    |   movel([0.078731, -1.406852, -2.551684, -0.753853, 1.570796, 1.649527],accel_mss,speed_ms,0,blend_radius_m)
    |   movel([0.077871, -1.407087, -2.551509, -0.753793, 1.570796, 1.648667],accel_mss,speed_ms,0,blend_radius_m)
    |   movel([0.077016, -1.407341, -2.551319, -0.753728, 1.570796, 1.647812],accel_mss,speed_ms,0,blend_radius_m)
    |   movel([0.076261, -1.407587, -2.551136, -0.753666, 1.570796, 1.647058],accel_mss,speed_ms,0,blend_radius_m)
    |   movel([0.075139, -1.407960, -2.550859, -0.753571, 1.570796, 1.645936],accel_mss,speed_ms,0,blend_radius_m)
    |   speed_ms = 0.003
    |   movel([0.075139, -1.411176, -2.552300, -0.748913, 1.570796, 1.645936],accel_mss,speed_ms,0,blend_radius_m)
    |   speed_ms = 0.007
    |   movel([0.074668, -1.411273, -2.552227, -0.748889, 1.570796, 1.645464],accel_mss,speed_ms,0,blend_radius_m)
    |   movel([0.074481, -1.411194, -2.552286, -0.748909, 1.570796, 1.645278],accel_mss,speed_ms,0,blend_radius_m)
    |   movel([0.074467, -1.410958, -2.552463, -0.748968, 1.570796, 1.645263],accel_mss,speed_ms,0,blend_radius_m)
    |   movel([0.074692, -1.410622, -2.552715, -0.749052, 1.570796, 1.645489],accel_mss,speed_ms,0,blend_radius_m)
    |   movel([0.075140, -1.410315, -2.552945, -0.749129, 1.570796, 1.645937],accel_mss,speed_ms,0,blend_radius_m)
    |   movel([0.075912, -1.409983, -2.553193, -0.749213, 1.570796, 1.646708],accel_mss,speed_ms,0,blend_radius_m)
    |   movel([0.077256, -1.409535, -2.553528, -0.749326, 1.570796, 1.648052],accel_mss,speed_ms,0,blend_radius_m)
    |   movel([0.078806, -1.409077, -2.553870, -0.749442, 1.570796, 1.649603],accel_mss,speed_ms,0,blend_radius_m)
    |   movel([0.079979, -1.408805, -2.554073, -0.749511, 1.570796, 1.650775],accel_mss,speed_ms,0,blend_radius_m)
    |   movel([0.080824, -1.408690, -2.554159, -0.749540, 1.570796, 1.651621],accel_mss,speed_ms,0,blend_radius_m)
    |   movel([0.081268, -1.408772, -2.554098, -0.749519, 1.570796, 1.652064],accel_mss,speed_ms,0,blend_radius_m)
    |   movel([0.081447, -1.408903, -2.554000, -0.749486, 1.570796, 1.652243],accel_mss,speed_ms,0,blend_radius_m)
    |   movel([0.081473, -1.409173, -2.553798, -0.749418, 1.570796, 1.652269],accel_mss,speed_ms,0,blend_radius_m)
    |   movel([0.081179, -1.409435, -2.553602, -0.749351, 1.570796, 1.651975],accel_mss,speed_ms,0,blend_radius_m)
    |   movel([0.080823, -1.409552, -2.553515, -0.749322, 1.570796, 1.651619],accel_mss,speed_ms,0,blend_radius_m)
    |   movel([0.080297, -1.409695, -2.553409, -0.749286, 1.570796, 1.651093],accel_mss,speed_ms,0,blend_radius_m)
    |   movel([0.079504, -1.409881, -2.553270, -0.749239, 1.570796, 1.650301],accel_mss,speed_ms,0,blend_radius_m)
    |   movel([0.078731, -1.410072, -2.553127, -0.749191, 1.570796, 1.649527],accel_mss,speed_ms,0,blend_radius_m)
    |   movel([0.077871, -1.410306, -2.552951, -0.749132, 1.570796, 1.648667],accel_mss,speed_ms,0,blend_radius_m)
    |   movel([0.077016, -1.410560, -2.552762, -0.749068, 1.570796, 1.647812],accel_mss,speed_ms,0,blend_radius_m)
    |   movel([0.076261, -1.410805, -2.552578, -0.749006, 1.570796, 1.647058],accel_mss,speed_ms,0,blend_radius_m)
    |   movel([0.075139, -1.411176, -2.552300, -0.748913, 1.570796, 1.645936],accel_mss,speed_ms,0,blend_radius_m)
    |   speed_ms = 0.003
    |   movel([0.075139, -1.398436, -2.546485, -0.767469, 1.570796, 1.645936],accel_mss,speed_ms,0,blend_radius_m)
    |   speed_ms = 1.000
    |   movel([0.075139, -1.373952, -2.534460, -0.803977, 1.570796, 1.645936],accel_mss,speed_ms,0,blend_radius_m)
    |   movel([0.075519, -1.372021, -2.535826, -0.804542, 1.570796, 1.646315],accel_mss,speed_ms,0,blend_radius_m)
    |   movel([0.075519, -1.396541, -2.547875, -0.767973, 1.570796, 1.646315],accel_mss,speed_ms,0,blend_radius_m)
    |   speed_ms = 0.003
    |   movel([0.075519, -1.406080, -2.552258, -0.754051, 1.570796, 1.646315],accel_mss,speed_ms,0,blend_radius_m)
    |   speed_ms = 0.007
    |   movel([0.075126, -1.406076, -2.552261, -0.754052, 1.570796, 1.645923],accel_mss,speed_ms,0,blend_radius_m)
    |   movel([0.074945, -1.405955, -2.552351, -0.754083, 1.570796, 1.645741],accel_mss,speed_ms,0,blend_radius_m)
    |   movel([0.074905, -1.405527, -2.552669, -0.754193, 1.570796, 1.645701],accel_mss,speed_ms,0,blend_radius_m)
    |   movel([0.074901, -1.405141, -2.552955, -0.754293, 1.570796, 1.645697],accel_mss,speed_ms,0,blend_radius_m)
    |   movel([0.074910, -1.404710, -2.553275, -0.754404, 1.570796, 1.645707],accel_mss,speed_ms,0,blend_radius_m)
    |   movel([0.074938, -1.404075, -2.553745, -0.754569, 1.570796, 1.645734],accel_mss,speed_ms,0,blend_radius_m)
    |   movel([0.074975, -1.403788, -2.553958, -0.754644, 1.570796, 1.645771],accel_mss,speed_ms,0,blend_radius_m)
    |   movel([0.075148, -1.403554, -2.554131, -0.754705, 1.570796, 1.645944],accel_mss,speed_ms,0,blend_radius_m)
    |   movel([0.075346, -1.403676, -2.554040, -0.754673, 1.570796, 1.646142],accel_mss,speed_ms,0,blend_radius_m)
    |   movel([0.075432, -1.403876, -2.553893, -0.754621, 1.570796, 1.646229],accel_mss,speed_ms,0,blend_radius_m)
    |   movel([0.075542, -1.404111, -2.553718, -0.754559, 1.570796, 1.646338],accel_mss,speed_ms,0,blend_radius_m)
    |   movel([0.075676, -1.404370, -2.553527, -0.754492, 1.570796, 1.646472],accel_mss,speed_ms,0,blend_radius_m)
    |   movel([0.075914, -1.404778, -2.553224, -0.754387, 1.570796, 1.646711],accel_mss,speed_ms,0,blend_radius_m)
    |   movel([0.076091, -1.404951, -2.553096, -0.754342, 1.570796, 1.646887],accel_mss,speed_ms,0,blend_radius_m)
    |   movel([0.076338, -1.405044, -2.553027, -0.754318, 1.570796, 1.647135],accel_mss,speed_ms,0,blend_radius_m)
    |   movel([0.076878, -1.405129, -2.552964, -0.754296, 1.570796, 1.647674],accel_mss,speed_ms,0,blend_radius_m)
    |   movel([0.077216, -1.405165, -2.552937, -0.754286, 1.570796, 1.648012],accel_mss,speed_ms,0,blend_radius_m)
    |   movel([0.077528, -1.405191, -2.552918, -0.754280, 1.570796, 1.648324],accel_mss,speed_ms,0,blend_radius_m)
    |   movel([0.077792, -1.405202, -2.552910, -0.754277, 1.570796, 1.648589],accel_mss,speed_ms,0,blend_radius_m)
    |   movel([0.078078, -1.405163, -2.552939, -0.754287, 1.570796, 1.648874],accel_mss,speed_ms,0,blend_radius_m)
    |   movel([0.078293, -1.405186, -2.552922, -0.754281, 1.570796, 1.649090],accel_mss,speed_ms,0,blend_radius_m)
    |   movel([0.078458, -1.405300, -2.552837, -0.754252, 1.570796, 1.649254],accel_mss,speed_ms,0,blend_radius_m)
    |   movel([0.078022, -1.405459, -2.552719, -0.754211, 1.570796, 1.648818],accel_mss,speed_ms,0,blend_radius_m)
    |   movel([0.077584, -1.405591, -2.552621, -0.754177, 1.570796, 1.648380],accel_mss,speed_ms,0,blend_radius_m)
    |   movel([0.077076, -1.405736, -2.552513, -0.754139, 1.570796, 1.647873],accel_mss,speed_ms,0,blend_radius_m)
    |   movel([0.076136, -1.405975, -2.552336, -0.754078, 1.570796, 1.646933],accel_mss,speed_ms,0,blend_radius_m)
    |   movel([0.075519, -1.406080, -2.552258, -0.754051, 1.570796, 1.646315],accel_mss,speed_ms,0,blend_radius_m)
    |   speed_ms = 0.003
    |   movel([0.075519, -1.409302, -2.553702, -0.749385, 1.570796, 1.646315],accel_mss,speed_ms,0,blend_radius_m)
    |   speed_ms = 0.007
    |   movel([0.075126, -1.409298, -2.553705, -0.749386, 1.570796, 1.645923],accel_mss,speed_ms,0,blend_radius_m)
    |   movel([0.074945, -1.409177, -2.553795, -0.749417, 1.570796, 1.645741],accel_mss,speed_ms,0,blend_radius_m)
    |   movel([0.074905, -1.408750, -2.554114, -0.749525, 1.570796, 1.645701],accel_mss,speed_ms,0,blend_radius_m)
    |   movel([0.074901, -1.408365, -2.554401, -0.749623, 1.570796, 1.645697],accel_mss,speed_ms,0,blend_radius_m)
    |   movel([0.074910, -1.407935, -2.554721, -0.749732, 1.570796, 1.645707],accel_mss,speed_ms,0,blend_radius_m)
    |   movel([0.074938, -1.407303, -2.555192, -0.749894, 1.570796, 1.645734],accel_mss,speed_ms,0,blend_radius_m)
    |   movel([0.074975, -1.407016, -2.555406, -0.749967, 1.570796, 1.645771],accel_mss,speed_ms,0,blend_radius_m)
    |   movel([0.075148, -1.406782, -2.555579, -0.750027, 1.570796, 1.645944],accel_mss,speed_ms,0,blend_radius_m)
    |   movel([0.075346, -1.406905, -2.555488, -0.749996, 1.570796, 1.646142],accel_mss,speed_ms,0,blend_radius_m)
    |   movel([0.075432, -1.407104, -2.555340, -0.749945, 1.570796, 1.646229],accel_mss,speed_ms,0,blend_radius_m)
    |   movel([0.075542, -1.407338, -2.555166, -0.749885, 1.570796, 1.646338],accel_mss,speed_ms,0,blend_radius_m)
    |   movel([0.075676, -1.407596, -2.554974, -0.749819, 1.570796, 1.646472],accel_mss,speed_ms,0,blend_radius_m)
    |   movel([0.075914, -1.408003, -2.554671, -0.749715, 1.570796, 1.646711],accel_mss,speed_ms,0,blend_radius_m)
    |   movel([0.076091, -1.408176, -2.554542, -0.749671, 1.570796, 1.646887],accel_mss,speed_ms,0,blend_radius_m)
    |   movel([0.076338, -1.408268, -2.554473, -0.749647, 1.570796, 1.647135],accel_mss,speed_ms,0,blend_radius_m)
    |   movel([0.076878, -1.408353, -2.554410, -0.749626, 1.570796, 1.647674],accel_mss,speed_ms,0,blend_radius_m)
    |   movel([0.077216, -1.408390, -2.554383, -0.749616, 1.570796, 1.648012],accel_mss,speed_ms,0,blend_radius_m)
    |   movel([0.077528, -1.408415, -2.554364, -0.749610, 1.570796, 1.648324],accel_mss,speed_ms,0,blend_radius_m)
    |   movel([0.077792, -1.408426, -2.554356, -0.749607, 1.570796, 1.648589],accel_mss,speed_ms,0,blend_radius_m)
    |   movel([0.078078, -1.408387, -2.554385, -0.749617, 1.570796, 1.648874],accel_mss,speed_ms,0,blend_radius_m)
    |   movel([0.078293, -1.408410, -2.554368, -0.749611, 1.570796, 1.649090],accel_mss,speed_ms,0,blend_radius_m)
    |   movel([0.078458, -1.408524, -2.554282, -0.749582, 1.570796, 1.649254],accel_mss,speed_ms,0,blend_radius_m)
    |   movel([0.078022, -1.408683, -2.554164, -0.749542, 1.570796, 1.648818],accel_mss,speed_ms,0,blend_radius_m)
    |   movel([0.077584, -1.408814, -2.554067, -0.749509, 1.570796, 1.648380],accel_mss,speed_ms,0,blend_radius_m)
    |   movel([0.077076, -1.408959, -2.553958, -0.749472, 1.570796, 1.647873],accel_mss,speed_ms,0,blend_radius_m)
    |   movel([0.076136, -1.409198, -2.553780, -0.749411, 1.570796, 1.646933],accel_mss,speed_ms,0,blend_radius_m)
    |   movel([0.075519, -1.409302, -2.553702, -0.749385, 1.570796, 1.646315],accel_mss,speed_ms,0,blend_radius_m)
    |   speed_ms = 0.003
    |   movel([0.075519, -1.396541, -2.547875, -0.767973, 1.570796, 1.646315],accel_mss,speed_ms,0,blend_radius_m)
    |   speed_ms = 1.000
    |   movel([0.075519, -1.372021, -2.535826, -0.804542, 1.570796, 1.646315],accel_mss,speed_ms,0,blend_radius_m)
    |   movel([0.077083, -1.370467, -2.536922, -0.805000, 1.570796, 1.647879],accel_mss,speed_ms,0,blend_radius_m)
    |   movel([0.077083, -1.395016, -2.548990, -0.768383, 1.570796, 1.647879],accel_mss,speed_ms,0,blend_radius_m)
    |   speed_ms = 0.003
    |   movel([0.077083, -1.404567, -2.553381, -0.754441, 1.570796, 1.647879],accel_mss,speed_ms,0,blend_radius_m)
    |   speed_ms = 0.007
    |   movel([0.076403, -1.404193, -2.553658, -0.754538, 1.570796, 1.647199],accel_mss,speed_ms,0,blend_radius_m)
    |   movel([0.076021, -1.403445, -2.554211, -0.754733, 1.570796, 1.646818],accel_mss,speed_ms,0,blend_radius_m)
    |   movel([0.075316, -1.401677, -2.555516, -0.755196, 1.570796, 1.646112],accel_mss,speed_ms,0,blend_radius_m)
    |   movel([0.074634, -1.399869, -2.556846, -0.755675, 1.570796, 1.645431],accel_mss,speed_ms,0,blend_radius_m)
    |   movel([0.074243, -1.398639, -2.557747, -0.756003, 1.570796, 1.645039],accel_mss,speed_ms,0,blend_radius_m)
    |   movel([0.074191, -1.398445, -2.557889, -0.756055, 1.570796, 1.644987],accel_mss,speed_ms,0,blend_radius_m)
    |   movel([0.074083, -1.398061, -2.558171, -0.756158, 1.570796, 1.644879],accel_mss,speed_ms,0,blend_radius_m)
    |   movel([0.073955, -1.397607, -2.558503, -0.756280, 1.570796, 1.644752],accel_mss,speed_ms,0,blend_radius_m)
    |   movel([0.073822, -1.397131, -2.558850, -0.756408, 1.570796, 1.644618],accel_mss,speed_ms,0,blend_radius_m)
    |   movel([0.073030, -1.393944, -2.561169, -0.757276, 1.570796, 1.643826],accel_mss,speed_ms,0,blend_radius_m)
    |   movel([0.072490, -1.390932, -2.563348, -0.758110, 1.570796, 1.643286],accel_mss,speed_ms,0,blend_radius_m)
    |   movel([0.072193, -1.387994, -2.565460, -0.758936, 1.570796, 1.642990],accel_mss,speed_ms,0,blend_radius_m)
    |   movel([0.072126, -1.385031, -2.567577, -0.759781, 1.570796, 1.642923],accel_mss,speed_ms,0,blend_radius_m)
    |   movel([0.072151, -1.383881, -2.568396, -0.760113, 1.570796, 1.642947],accel_mss,speed_ms,0,blend_radius_m)
    |   movel([0.072187, -1.383304, -2.568805, -0.760280, 1.570796, 1.642984],accel_mss,speed_ms,0,blend_radius_m)
    |   movel([0.072246, -1.382955, -2.569053, -0.760381, 1.570796, 1.643042],accel_mss,speed_ms,0,blend_radius_m)
    |   movel([0.072513, -1.382648, -2.569271, -0.760471, 1.570796, 1.643309],accel_mss,speed_ms,0,blend_radius_m)
    |   movel([0.073127, -1.382500, -2.569376, -0.760513, 1.570796, 1.643923],accel_mss,speed_ms,0,blend_radius_m)
    |   movel([0.073892, -1.382409, -2.569440, -0.760540, 1.570796, 1.644689],accel_mss,speed_ms,0,blend_radius_m)
    |   movel([0.079022, -1.381656, -2.569973, -0.760760, 1.570796, 1.649818],accel_mss,speed_ms,0,blend_radius_m)
    |   movel([0.084810, -1.380457, -2.570821, -0.761111, 1.570796, 1.655606],accel_mss,speed_ms,0,blend_radius_m)
    |   movel([0.090456, -1.379003, -2.571845, -0.761540, 1.570796, 1.661253],accel_mss,speed_ms,0,blend_radius_m)
    |   movel([0.095111, -1.377468, -2.572924, -0.761997, 1.570796, 1.665908],accel_mss,speed_ms,0,blend_radius_m)
    |   movel([0.097708, -1.376448, -2.573639, -0.762302, 1.570796, 1.668504],accel_mss,speed_ms,0,blend_radius_m)
    |   movel([0.100378, -1.375309, -2.574435, -0.762644, 1.570796, 1.671174],accel_mss,speed_ms,0,blend_radius_m)
    |   movel([0.102904, -1.374151, -2.575243, -0.762994, 1.570796, 1.673700],accel_mss,speed_ms,0,blend_radius_m)
    |   movel([0.105045, -1.373074, -2.575993, -0.763322, 1.570796, 1.675841],accel_mss,speed_ms,0,blend_radius_m)
    |   movel([0.105543, -1.372819, -2.576171, -0.763400, 1.570796, 1.676340],accel_mss,speed_ms,0,blend_radius_m)
    |   movel([0.105878, -1.372668, -2.576275, -0.763446, 1.570796, 1.676675],accel_mss,speed_ms,0,blend_radius_m)
    |   movel([0.106228, -1.372598, -2.576324, -0.763467, 1.570796, 1.677024],accel_mss,speed_ms,0,blend_radius_m)
    |   movel([0.106336, -1.372808, -2.576178, -0.763403, 1.570796, 1.677133],accel_mss,speed_ms,0,blend_radius_m)
    |   movel([0.106198, -1.374131, -2.575258, -0.763001, 1.570796, 1.676995],accel_mss,speed_ms,0,blend_radius_m)
    |   movel([0.105975, -1.375739, -2.574135, -0.762515, 1.570796, 1.676771],accel_mss,speed_ms,0,blend_radius_m)
    |   movel([0.105644, -1.377653, -2.572794, -0.761942, 1.570796, 1.676440],accel_mss,speed_ms,0,blend_radius_m)
    |   movel([0.104699, -1.381947, -2.569767, -0.760675, 1.570796, 1.675495],accel_mss,speed_ms,0,blend_radius_m)
    |   movel([0.103481, -1.386121, -2.566799, -0.759469, 1.570796, 1.674277],accel_mss,speed_ms,0,blend_radius_m)
    |   movel([0.102014, -1.390127, -2.563928, -0.758335, 1.570796, 1.672810],accel_mss,speed_ms,0,blend_radius_m)
    |   movel([0.100315, -1.393925, -2.561183, -0.757281, 1.570796, 1.671111],accel_mss,speed_ms,0,blend_radius_m)
    |   movel([0.099682, -1.395155, -2.560289, -0.756944, 1.570796, 1.670478],accel_mss,speed_ms,0,blend_radius_m)
    |   movel([0.098968, -1.396436, -2.559357, -0.756596, 1.570796, 1.669764],accel_mss,speed_ms,0,blend_radius_m)
    |   movel([0.098297, -1.397567, -2.558532, -0.756291, 1.570796, 1.669093],accel_mss,speed_ms,0,blend_radius_m)
    |   movel([0.097942, -1.398033, -2.558191, -0.756165, 1.570796, 1.668739],accel_mss,speed_ms,0,blend_radius_m)
    |   movel([0.097526, -1.398382, -2.557935, -0.756072, 1.570796, 1.668322],accel_mss,speed_ms,0,blend_radius_m)
    |   movel([0.096641, -1.398930, -2.557534, -0.755925, 1.570796, 1.667437],accel_mss,speed_ms,0,blend_radius_m)
    |   movel([0.095567, -1.399532, -2.557093, -0.755764, 1.570796, 1.666363],accel_mss,speed_ms,0,blend_radius_m)
    |   movel([0.094415, -1.400113, -2.556666, -0.755610, 1.570796, 1.665211],accel_mss,speed_ms,0,blend_radius_m)
    |   movel([0.091915, -1.401217, -2.555855, -0.755317, 1.570796, 1.662711],accel_mss,speed_ms,0,blend_radius_m)
    |   movel([0.089053, -1.402291, -2.555063, -0.755035, 1.570796, 1.659849],accel_mss,speed_ms,0,blend_radius_m)
    |   movel([0.086165, -1.403221, -2.554377, -0.754791, 1.570796, 1.656961],accel_mss,speed_ms,0,blend_radius_m)
    |   movel([0.083581, -1.403891, -2.553881, -0.754617, 1.570796, 1.654377],accel_mss,speed_ms,0,blend_radius_m)
    |   movel([0.080960, -1.404386, -2.553515, -0.754488, 1.570796, 1.651756],accel_mss,speed_ms,0,blend_radius_m)
    |   movel([0.078742, -1.404605, -2.553352, -0.754431, 1.570796, 1.649539],accel_mss,speed_ms,0,blend_radius_m)
    |   movel([0.077083, -1.404567, -2.553381, -0.754441, 1.570796, 1.647879],accel_mss,speed_ms,0,blend_radius_m)
    |   speed_ms = 0.003
    |   movel([0.077083, -1.407793, -2.554827, -0.749769, 1.570796, 1.647879],accel_mss,speed_ms,0,blend_radius_m)
    |   speed_ms = 0.007
    |   movel([0.076403, -1.407420, -2.555105, -0.749864, 1.570796, 1.647199],accel_mss,speed_ms,0,blend_radius_m)
    |   movel([0.076021, -1.406674, -2.555660, -0.750055, 1.570796, 1.646818],accel_mss,speed_ms,0,blend_radius_m)
    |   movel([0.075316, -1.404911, -2.556967, -0.750510, 1.570796, 1.646112],accel_mss,speed_ms,0,blend_radius_m)
    |   movel([0.074634, -1.403108, -2.558300, -0.750981, 1.570796, 1.645431],accel_mss,speed_ms,0,blend_radius_m)
    |   movel([0.074243, -1.401882, -2.559203, -0.751304, 1.570796, 1.645039],accel_mss,speed_ms,0,blend_radius_m)
    |   movel([0.074191, -1.401688, -2.559346, -0.751355, 1.570796, 1.644987],accel_mss,speed_ms,0,blend_radius_m)
    |   movel([0.074083, -1.401305, -2.559628, -0.751456, 1.570796, 1.644879],accel_mss,speed_ms,0,blend_radius_m)
    |   movel([0.073955, -1.400852, -2.559960, -0.751576, 1.570796, 1.644752],accel_mss,speed_ms,0,blend_radius_m)
    |   movel([0.073822, -1.400378, -2.560308, -0.751702, 1.570796, 1.644618],accel_mss,speed_ms,0,blend_radius_m)
    |   movel([0.073030, -1.397200, -2.562633, -0.752556, 1.570796, 1.643826],accel_mss,speed_ms,0,blend_radius_m)
    |   movel([0.072490, -1.394196, -2.564816, -0.753377, 1.570796, 1.643286],accel_mss,speed_ms,0,blend_radius_m)
    |   movel([0.072193, -1.391266, -2.566933, -0.754190, 1.570796, 1.642990],accel_mss,speed_ms,0,blend_radius_m)
    |   movel([0.072126, -1.388311, -2.569056, -0.755023, 1.570796, 1.642923],accel_mss,speed_ms,0,blend_radius_m)
    |   movel([0.072151, -1.387164, -2.569876, -0.755349, 1.570796, 1.642947],accel_mss,speed_ms,0,blend_radius_m)
    |   movel([0.072187, -1.386589, -2.570287, -0.755514, 1.570796, 1.642984],accel_mss,speed_ms,0,blend_radius_m)
    |   movel([0.072246, -1.386241, -2.570535, -0.755613, 1.570796, 1.643042],accel_mss,speed_ms,0,blend_radius_m)
    |   movel([0.072513, -1.385934, -2.570753, -0.755701, 1.570796, 1.643309],accel_mss,speed_ms,0,blend_radius_m)
    |   movel([0.073127, -1.385787, -2.570858, -0.755744, 1.570796, 1.643923],accel_mss,speed_ms,0,blend_radius_m)
    |   movel([0.073892, -1.385697, -2.570922, -0.755770, 1.570796, 1.644689],accel_mss,speed_ms,0,blend_radius_m)
    |   movel([0.079022, -1.384945, -2.571457, -0.755986, 1.570796, 1.649818],accel_mss,speed_ms,0,blend_radius_m)
    |   movel([0.084810, -1.383749, -2.572307, -0.756333, 1.570796, 1.655606],accel_mss,speed_ms,0,blend_radius_m)
    |   movel([0.090456, -1.382300, -2.573334, -0.756755, 1.570796, 1.661253],accel_mss,speed_ms,0,blend_radius_m)
    |   movel([0.095111, -1.380769, -2.574415, -0.757205, 1.570796, 1.665908],accel_mss,speed_ms,0,blend_radius_m)
    |   movel([0.097708, -1.379752, -2.575132, -0.757506, 1.570796, 1.668504],accel_mss,speed_ms,0,blend_radius_m)
    |   movel([0.100378, -1.378616, -2.575930, -0.757843, 1.570796, 1.671174],accel_mss,speed_ms,0,blend_radius_m)
    |   movel([0.102904, -1.377461, -2.576739, -0.758188, 1.570796, 1.673700],accel_mss,speed_ms,0,blend_radius_m)
    |   movel([0.105045, -1.376387, -2.577491, -0.758511, 1.570796, 1.675841],accel_mss,speed_ms,0,blend_radius_m)
    |   movel([0.105543, -1.376132, -2.577669, -0.758588, 1.570796, 1.676340],accel_mss,speed_ms,0,blend_radius_m)
    |   movel([0.105878, -1.375982, -2.577774, -0.758633, 1.570796, 1.676675],accel_mss,speed_ms,0,blend_radius_m)
    |   movel([0.106228, -1.375912, -2.577822, -0.758654, 1.570796, 1.677024],accel_mss,speed_ms,0,blend_radius_m)
    |   movel([0.106336, -1.376121, -2.577677, -0.758591, 1.570796, 1.677133],accel_mss,speed_ms,0,blend_radius_m)
    |   movel([0.106198, -1.377441, -2.576754, -0.758194, 1.570796, 1.676995],accel_mss,speed_ms,0,blend_radius_m)
    |   movel([0.105975, -1.379044, -2.575629, -0.757716, 1.570796, 1.676771],accel_mss,speed_ms,0,blend_radius_m)
    |   movel([0.105644, -1.380953, -2.574285, -0.757151, 1.570796, 1.676440],accel_mss,speed_ms,0,blend_radius_m)
    |   movel([0.104699, -1.385235, -2.571251, -0.755903, 1.570796, 1.675495],accel_mss,speed_ms,0,blend_radius_m)
    |   movel([0.103481, -1.389398, -2.568276, -0.754715, 1.570796, 1.674277],accel_mss,speed_ms,0,blend_radius_m)
    |   movel([0.102014, -1.393393, -2.565398, -0.753598, 1.570796, 1.672810],accel_mss,speed_ms,0,blend_radius_m)
    |   movel([0.100315, -1.397181, -2.562647, -0.752561, 1.570796, 1.671111],accel_mss,speed_ms,0,blend_radius_m)
    |   movel([0.099682, -1.398408, -2.561751, -0.752230, 1.570796, 1.670478],accel_mss,speed_ms,0,blend_radius_m)
    |   movel([0.098968, -1.399685, -2.560817, -0.751887, 1.570796, 1.669764],accel_mss,speed_ms,0,blend_radius_m)
    |   movel([0.098297, -1.400812, -2.559990, -0.751587, 1.570796, 1.669093],accel_mss,speed_ms,0,blend_radius_m)
    |   movel([0.097942, -1.401278, -2.559648, -0.751464, 1.570796, 1.668739],accel_mss,speed_ms,0,blend_radius_m)
    |   movel([0.097526, -1.401625, -2.559392, -0.751372, 1.570796, 1.668322],accel_mss,speed_ms,0,blend_radius_m)
    |   movel([0.096641, -1.402172, -2.558990, -0.751227, 1.570796, 1.667437],accel_mss,speed_ms,0,blend_radius_m)
    |   movel([0.095567, -1.402772, -2.558548, -0.751069, 1.570796, 1.666363],accel_mss,speed_ms,0,blend_radius_m)
    |   movel([0.094415, -1.403352, -2.558120, -0.750917, 1.570796, 1.665211],accel_mss,speed_ms,0,blend_radius_m)
    |   movel([0.091915, -1.404453, -2.557307, -0.750630, 1.570796, 1.662711],accel_mss,speed_ms,0,blend_radius_m)
    |   movel([0.089053, -1.405523, -2.556514, -0.750352, 1.570796, 1.659849],accel_mss,speed_ms,0,blend_radius_m)
    |   movel([0.086165, -1.406451, -2.555826, -0.750113, 1.570796, 1.656961],accel_mss,speed_ms,0,blend_radius_m)
    |   movel([0.083581, -1.407119, -2.555329, -0.749941, 1.570796, 1.654377],accel_mss,speed_ms,0,blend_radius_m)
    |   movel([0.080960, -1.407612, -2.554962, -0.749815, 1.570796, 1.651756],accel_mss,speed_ms,0,blend_radius_m)
    |   movel([0.078742, -1.407831, -2.554799, -0.749759, 1.570796, 1.649539],accel_mss,speed_ms,0,blend_radius_m)
    |   movel([0.077083, -1.407793, -2.554827, -0.749769, 1.570796, 1.647879],accel_mss,speed_ms,0,blend_radius_m)
    |   speed_ms = 0.003
    |   movel([0.077083, -1.395016, -2.548990, -0.768383, 1.570796, 1.647879],accel_mss,speed_ms,0,blend_radius_m)
    |   speed_ms = 1.000
    |   movel([0.077083, -1.370467, -2.536922, -0.805000, 1.570796, 1.647879],accel_mss,speed_ms,0,blend_radius_m)
    |   movel([0.095608, -1.366022, -2.540038, -0.806329, 1.570796, 1.666405],accel_mss,speed_ms,0,blend_radius_m)
    |   movel([0.095608, -1.390653, -2.552162, -0.769574, 1.570796, 1.666405],accel_mss,speed_ms,0,blend_radius_m)
    |   speed_ms = 0.003
    |   movel([0.095608, -1.400240, -2.556573, -0.755576, 1.570796, 1.666405],accel_mss,speed_ms,0,blend_radius_m)
    |   speed_ms = 0.007
    |   movel([0.096849, -1.399375, -2.557208, -0.755806, 1.570796, 1.667646],accel_mss,speed_ms,0,blend_radius_m)
    |   movel([0.097726, -1.398829, -2.557608, -0.755952, 1.570796, 1.668522],accel_mss,speed_ms,0,blend_radius_m)
    |   movel([0.098243, -1.398433, -2.557898, -0.756058, 1.570796, 1.669039],accel_mss,speed_ms,0,blend_radius_m)
    |   movel([0.098617, -1.398025, -2.558196, -0.756167, 1.570796, 1.669413],accel_mss,speed_ms,0,blend_radius_m)
    |   movel([0.098982, -1.397470, -2.558602, -0.756317, 1.570796, 1.669778],accel_mss,speed_ms,0,blend_radius_m)
    |   movel([0.099332, -1.396906, -2.559014, -0.756469, 1.570796, 1.670128],accel_mss,speed_ms,0,blend_radius_m)
    |   movel([0.099610, -1.396984, -2.558957, -0.756448, 1.570796, 1.670406],accel_mss,speed_ms,0,blend_radius_m)
    |   movel([0.099548, -1.397682, -2.558447, -0.756260, 1.570796, 1.670344],accel_mss,speed_ms,0,blend_radius_m)
    |   movel([0.099497, -1.398045, -2.558182, -0.756162, 1.570796, 1.670293],accel_mss,speed_ms,0,blend_radius_m)
    |   movel([0.099431, -1.398388, -2.557931, -0.756070, 1.570796, 1.670227],accel_mss,speed_ms,0,blend_radius_m)
    |   movel([0.099362, -1.398676, -2.557720, -0.755993, 1.570796, 1.670158],accel_mss,speed_ms,0,blend_radius_m)
    |   movel([0.099054, -1.399064, -2.557436, -0.755889, 1.570796, 1.669851],accel_mss,speed_ms,0,blend_radius_m)
    |   movel([0.098629, -1.399306, -2.557259, -0.755824, 1.570796, 1.669425],accel_mss,speed_ms,0,blend_radius_m)
    |   movel([0.097967, -1.399580, -2.557058, -0.755751, 1.570796, 1.668764],accel_mss,speed_ms,0,blend_radius_m)
    |   movel([0.096936, -1.399930, -2.556801, -0.755658, 1.570796, 1.667732],accel_mss,speed_ms,0,blend_radius_m)
    |   movel([0.095753, -1.400300, -2.556529, -0.755560, 1.570796, 1.666550],accel_mss,speed_ms,0,blend_radius_m)
    |   speed_ms = 0.003
    |   movel([0.095608, -1.403478, -2.558027, -0.750884, 1.570796, 1.666405],accel_mss,speed_ms,0,blend_radius_m)
    |   speed_ms = 0.007
    |   movel([0.096849, -1.402615, -2.558663, -0.751110, 1.570796, 1.667646],accel_mss,speed_ms,0,blend_radius_m)
    |   movel([0.097726, -1.402072, -2.559064, -0.751254, 1.570796, 1.668522],accel_mss,speed_ms,0,blend_radius_m)
    |   movel([0.098243, -1.401677, -2.559354, -0.751358, 1.570796, 1.669039],accel_mss,speed_ms,0,blend_radius_m)
    |   movel([0.098617, -1.401270, -2.559654, -0.751466, 1.570796, 1.669413],accel_mss,speed_ms,0,blend_radius_m)
    |   movel([0.098982, -1.400716, -2.560060, -0.751613, 1.570796, 1.669778],accel_mss,speed_ms,0,blend_radius_m)
    |   movel([0.099332, -1.400154, -2.560473, -0.751762, 1.570796, 1.670128],accel_mss,speed_ms,0,blend_radius_m)
    |   movel([0.099610, -1.400231, -2.560416, -0.751742, 1.570796, 1.670406],accel_mss,speed_ms,0,blend_radius_m)
    |   movel([0.099548, -1.400927, -2.559905, -0.751556, 1.570796, 1.670344],accel_mss,speed_ms,0,blend_radius_m)
    |   movel([0.099497, -1.401290, -2.559639, -0.751460, 1.570796, 1.670293],accel_mss,speed_ms,0,blend_radius_m)
    |   movel([0.099431, -1.401631, -2.559388, -0.751370, 1.570796, 1.670227],accel_mss,speed_ms,0,blend_radius_m)
    |   movel([0.099362, -1.401919, -2.559176, -0.751294, 1.570796, 1.670158],accel_mss,speed_ms,0,blend_radius_m)
    |   movel([0.099054, -1.402305, -2.558892, -0.751192, 1.570796, 1.669851],accel_mss,speed_ms,0,blend_radius_m)
    |   movel([0.098629, -1.402547, -2.558714, -0.751128, 1.570796, 1.669425],accel_mss,speed_ms,0,blend_radius_m)
    |   movel([0.097967, -1.402820, -2.558513, -0.751057, 1.570796, 1.668764],accel_mss,speed_ms,0,blend_radius_m)
    |   movel([0.096936, -1.403169, -2.558255, -0.750965, 1.570796, 1.667732],accel_mss,speed_ms,0,blend_radius_m)
    |   movel([0.095753, -1.403538, -2.557983, -0.750868, 1.570796, 1.666550],accel_mss,speed_ms,0,blend_radius_m)
    |   speed_ms = 0.003
    |   movel([0.095608, -1.390653, -2.552162, -0.769574, 1.570796, 1.666405],accel_mss,speed_ms,0,blend_radius_m)
    |   speed_ms = 1.000
    |   movel([0.095608, -1.366022, -2.540038, -0.806329, 1.570796, 1.666405],accel_mss,speed_ms,0,blend_radius_m)
    |   movel([0.095795, -1.366921, -2.539410, -0.806058, 1.570796, 1.666591],accel_mss,speed_ms,0,blend_radius_m)
    |   movel([0.095795, -1.391535, -2.551523, -0.769331, 1.570796, 1.666591],accel_mss,speed_ms,0,blend_radius_m)
    |   speed_ms = 0.003
    |   movel([0.095795, -1.401115, -2.555930, -0.755344, 1.570796, 1.666591],accel_mss,speed_ms,0,blend_radius_m)
    |   speed_ms = 0.007
    |   movel([0.097270, -1.400757, -2.556193, -0.755439, 1.570796, 1.668067],accel_mss,speed_ms,0,blend_radius_m)
    |   movel([0.098200, -1.400570, -2.556331, -0.755488, 1.570796, 1.668996],accel_mss,speed_ms,0,blend_radius_m)
    |   movel([0.098654, -1.400503, -2.556380, -0.755506, 1.570796, 1.669451],accel_mss,speed_ms,0,blend_radius_m)
    |   movel([0.098932, -1.400512, -2.556374, -0.755504, 1.570796, 1.669729],accel_mss,speed_ms,0,blend_radius_m)
    |   movel([0.099151, -1.400587, -2.556318, -0.755484, 1.570796, 1.669947],accel_mss,speed_ms,0,blend_radius_m)
    |   movel([0.099338, -1.400726, -2.556216, -0.755447, 1.570796, 1.670134],accel_mss,speed_ms,0,blend_radius_m)
    |   movel([0.099360, -1.401005, -2.556011, -0.755373, 1.570796, 1.670156],accel_mss,speed_ms,0,blend_radius_m)
    |   movel([0.099047, -1.401276, -2.555811, -0.755302, 1.570796, 1.669844],accel_mss,speed_ms,0,blend_radius_m)
    |   movel([0.098716, -1.401382, -2.555733, -0.755274, 1.570796, 1.669513],accel_mss,speed_ms,0,blend_radius_m)
    |   movel([0.098213, -1.401508, -2.555640, -0.755240, 1.570796, 1.669009],accel_mss,speed_ms,0,blend_radius_m)
    |   movel([0.097407, -1.401678, -2.555515, -0.755196, 1.570796, 1.668203],accel_mss,speed_ms,0,blend_radius_m)
    |   movel([0.096581, -1.401860, -2.555381, -0.755148, 1.570796, 1.667377],accel_mss,speed_ms,0,blend_radius_m)
    |   movel([0.095800, -1.402058, -2.555235, -0.755096, 1.570796, 1.666597],accel_mss,speed_ms,0,blend_radius_m)
    |   movel([0.095027, -1.402282, -2.555070, -0.755037, 1.570796, 1.665823],accel_mss,speed_ms,0,blend_radius_m)
    |   movel([0.094218, -1.402546, -2.554876, -0.754968, 1.570796, 1.665014],accel_mss,speed_ms,0,blend_radius_m)
    |   movel([0.093145, -1.402897, -2.554616, -0.754876, 1.570796, 1.663941],accel_mss,speed_ms,0,blend_radius_m)
    |   movel([0.092652, -1.403004, -2.554537, -0.754848, 1.570796, 1.663448],accel_mss,speed_ms,0,blend_radius_m)
    |   movel([0.092424, -1.402949, -2.554578, -0.754862, 1.570796, 1.663220],accel_mss,speed_ms,0,blend_radius_m)
    |   movel([0.092353, -1.402753, -2.554722, -0.754913, 1.570796, 1.663149],accel_mss,speed_ms,0,blend_radius_m)
    |   movel([0.092529, -1.402431, -2.554960, -0.754998, 1.570796, 1.663326],accel_mss,speed_ms,0,blend_radius_m)
    |   movel([0.093124, -1.402001, -2.555277, -0.755111, 1.570796, 1.663921],accel_mss,speed_ms,0,blend_radius_m)
    |   movel([0.094351, -1.401555, -2.555606, -0.755228, 1.570796, 1.665147],accel_mss,speed_ms,0,blend_radius_m)
    |   movel([0.095795, -1.401115, -2.555930, -0.755344, 1.570796, 1.666591],accel_mss,speed_ms,0,blend_radius_m)
    |   speed_ms = 0.003
    |   movel([0.095795, -1.404350, -2.557382, -0.750656, 1.570796, 1.666591],accel_mss,speed_ms,0,blend_radius_m)
    |   speed_ms = 0.007
    |   movel([0.097270, -1.403994, -2.557646, -0.750749, 1.570796, 1.668067],accel_mss,speed_ms,0,blend_radius_m)
    |   movel([0.098200, -1.403807, -2.557784, -0.750798, 1.570796, 1.668996],accel_mss,speed_ms,0,blend_radius_m)
    |   movel([0.098654, -1.403741, -2.557833, -0.750815, 1.570796, 1.669451],accel_mss,speed_ms,0,blend_radius_m)
    |   movel([0.098932, -1.403749, -2.557827, -0.750813, 1.570796, 1.669729],accel_mss,speed_ms,0,blend_radius_m)
    |   movel([0.099151, -1.403824, -2.557771, -0.750794, 1.570796, 1.669947],accel_mss,speed_ms,0,blend_radius_m)
    |   movel([0.099338, -1.403962, -2.557669, -0.750758, 1.570796, 1.670134],accel_mss,speed_ms,0,blend_radius_m)
    |   movel([0.099360, -1.404241, -2.557463, -0.750685, 1.570796, 1.670156],accel_mss,speed_ms,0,blend_radius_m)
    |   movel([0.099047, -1.404511, -2.557263, -0.750614, 1.570796, 1.669844],accel_mss,speed_ms,0,blend_radius_m)
    |   movel([0.098716, -1.404617, -2.557185, -0.750587, 1.570796, 1.669513],accel_mss,speed_ms,0,blend_radius_m)
    |   movel([0.098213, -1.404743, -2.557092, -0.750554, 1.570796, 1.669009],accel_mss,speed_ms,0,blend_radius_m)
    |   movel([0.097407, -1.404912, -2.556967, -0.750510, 1.570796, 1.668203],accel_mss,speed_ms,0,blend_radius_m)
    |   movel([0.096581, -1.405094, -2.556832, -0.750463, 1.570796, 1.667377],accel_mss,speed_ms,0,blend_radius_m)
    |   movel([0.095800, -1.405291, -2.556686, -0.750412, 1.570796, 1.666597],accel_mss,speed_ms,0,blend_radius_m)
    |   movel([0.095027, -1.405514, -2.556521, -0.750354, 1.570796, 1.665823],accel_mss,speed_ms,0,blend_radius_m)
    |   movel([0.094218, -1.405777, -2.556325, -0.750286, 1.570796, 1.665014],accel_mss,speed_ms,0,blend_radius_m)
    |   movel([0.093145, -1.406127, -2.556066, -0.750196, 1.570796, 1.663941],accel_mss,speed_ms,0,blend_radius_m)
    |   movel([0.092652, -1.406234, -2.555986, -0.750168, 1.570796, 1.663448],accel_mss,speed_ms,0,blend_radius_m)
    |   movel([0.092424, -1.406179, -2.556027, -0.750182, 1.570796, 1.663220],accel_mss,speed_ms,0,blend_radius_m)
    |   movel([0.092353, -1.405984, -2.556172, -0.750233, 1.570796, 1.663149],accel_mss,speed_ms,0,blend_radius_m)
    |   movel([0.092529, -1.405663, -2.556410, -0.750316, 1.570796, 1.663326],accel_mss,speed_ms,0,blend_radius_m)
    |   movel([0.093124, -1.405234, -2.556728, -0.750427, 1.570796, 1.663921],accel_mss,speed_ms,0,blend_radius_m)
    |   movel([0.094351, -1.404789, -2.557058, -0.750542, 1.570796, 1.665147],accel_mss,speed_ms,0,blend_radius_m)
    |   movel([0.095795, -1.404350, -2.557382, -0.750656, 1.570796, 1.666591],accel_mss,speed_ms,0,blend_radius_m)
    |   speed_ms = 0.003
    |   movel([0.095795, -1.391535, -2.551523, -0.769331, 1.570796, 1.666591],accel_mss,speed_ms,0,blend_radius_m)
    |   speed_ms = 1.000
    |   movel([0.095795, -1.366921, -2.539410, -0.806058, 1.570796, 1.666591],accel_mss,speed_ms,0,blend_radius_m)
    |   movel([0.095058, -1.368794, -2.538098, -0.805497, 1.570796, 1.665854],accel_mss,speed_ms,0,blend_radius_m)
    |   movel([0.095058, -1.393374, -2.550187, -0.768828, 1.570796, 1.665854],accel_mss,speed_ms,0,blend_radius_m)
    |   speed_ms = 0.003
    |   movel([0.095058, -1.402939, -2.554585, -0.754865, 1.570796, 1.665854],accel_mss,speed_ms,0,blend_radius_m)
    |   speed_ms = 0.007
    |   movel([0.096957, -1.402395, -2.554986, -0.755007, 1.570796, 1.667754],accel_mss,speed_ms,0,blend_radius_m)
    |   movel([0.098037, -1.402157, -2.555162, -0.755070, 1.570796, 1.668833],accel_mss,speed_ms,0,blend_radius_m)
    |   movel([0.098676, -1.402118, -2.555191, -0.755080, 1.570796, 1.669473],accel_mss,speed_ms,0,blend_radius_m)
    |   movel([0.099066, -1.402259, -2.555087, -0.755043, 1.570796, 1.669862],accel_mss,speed_ms,0,blend_radius_m)
    |   movel([0.099131, -1.402534, -2.554884, -0.754971, 1.570796, 1.669927],accel_mss,speed_ms,0,blend_radius_m)
    |   movel([0.098905, -1.402879, -2.554629, -0.754881, 1.570796, 1.669701],accel_mss,speed_ms,0,blend_radius_m)
    |   movel([0.098649, -1.402995, -2.554544, -0.754850, 1.570796, 1.669445],accel_mss,speed_ms,0,blend_radius_m)
    |   movel([0.098218, -1.403073, -2.554486, -0.754830, 1.570796, 1.669014],accel_mss,speed_ms,0,blend_radius_m)
    |   movel([0.097382, -1.403224, -2.554375, -0.754791, 1.570796, 1.668179],accel_mss,speed_ms,0,blend_radius_m)
    |   movel([0.095577, -1.403702, -2.554021, -0.754666, 1.570796, 1.666373],accel_mss,speed_ms,0,blend_radius_m)
    |   movel([0.093763, -1.404215, -2.553642, -0.754533, 1.570796, 1.664560],accel_mss,speed_ms,0,blend_radius_m)
    |   movel([0.092999, -1.404503, -2.553428, -0.754458, 1.570796, 1.663795],accel_mss,speed_ms,0,blend_radius_m)
    |   movel([0.092709, -1.404629, -2.553335, -0.754425, 1.570796, 1.663506],accel_mss,speed_ms,0,blend_radius_m)
    |   movel([0.092398, -1.404692, -2.553288, -0.754409, 1.570796, 1.663195],accel_mss,speed_ms,0,blend_radius_m)
    |   movel([0.092200, -1.404501, -2.553429, -0.754458, 1.570796, 1.662996],accel_mss,speed_ms,0,blend_radius_m)
    |   movel([0.092240, -1.404260, -2.553608, -0.754521, 1.570796, 1.663036],accel_mss,speed_ms,0,blend_radius_m)
    |   movel([0.092394, -1.403991, -2.553808, -0.754591, 1.570796, 1.663190],accel_mss,speed_ms,0,blend_radius_m)
    |   movel([0.092628, -1.403768, -2.553972, -0.754649, 1.570796, 1.663424],accel_mss,speed_ms,0,blend_radius_m)
    |   movel([0.093075, -1.403542, -2.554139, -0.754707, 1.570796, 1.663871],accel_mss,speed_ms,0,blend_radius_m)
    |   movel([0.095058, -1.402939, -2.554585, -0.754865, 1.570796, 1.665854],accel_mss,speed_ms,0,blend_radius_m)
    |   speed_ms = 0.003
    |   movel([0.095058, -1.406170, -2.556034, -0.750185, 1.570796, 1.665854],accel_mss,speed_ms,0,blend_radius_m)
    |   speed_ms = 0.007
    |   movel([0.096957, -1.405627, -2.556437, -0.750325, 1.570796, 1.667754],accel_mss,speed_ms,0,blend_radius_m)
    |   movel([0.098037, -1.405390, -2.556613, -0.750386, 1.570796, 1.668833],accel_mss,speed_ms,0,blend_radius_m)
    |   movel([0.098676, -1.405351, -2.556641, -0.750396, 1.570796, 1.669473],accel_mss,speed_ms,0,blend_radius_m)
    |   movel([0.099066, -1.405491, -2.556537, -0.750360, 1.570796, 1.669862],accel_mss,speed_ms,0,blend_radius_m)
    |   movel([0.099131, -1.405766, -2.556334, -0.750289, 1.570796, 1.669927],accel_mss,speed_ms,0,blend_radius_m)
    |   movel([0.098905, -1.406110, -2.556079, -0.750200, 1.570796, 1.669701],accel_mss,speed_ms,0,blend_radius_m)
    |   movel([0.098649, -1.406225, -2.555993, -0.750171, 1.570796, 1.669445],accel_mss,speed_ms,0,blend_radius_m)
    |   movel([0.098218, -1.406303, -2.555935, -0.750151, 1.570796, 1.669014],accel_mss,speed_ms,0,blend_radius_m)
    |   movel([0.097382, -1.406453, -2.555824, -0.750112, 1.570796, 1.668179],accel_mss,speed_ms,0,blend_radius_m)
    |   movel([0.095577, -1.406930, -2.555469, -0.749989, 1.570796, 1.666373],accel_mss,speed_ms,0,blend_radius_m)
    |   movel([0.093763, -1.407442, -2.555089, -0.749858, 1.570796, 1.664560],accel_mss,speed_ms,0,blend_radius_m)
    |   movel([0.092999, -1.407729, -2.554875, -0.749785, 1.570796, 1.663795],accel_mss,speed_ms,0,blend_radius_m)
    |   movel([0.092709, -1.407855, -2.554782, -0.749753, 1.570796, 1.663506],accel_mss,speed_ms,0,blend_radius_m)
    |   movel([0.092398, -1.407917, -2.554735, -0.749737, 1.570796, 1.663195],accel_mss,speed_ms,0,blend_radius_m)
    |   movel([0.092200, -1.407728, -2.554876, -0.749785, 1.570796, 1.662996],accel_mss,speed_ms,0,blend_radius_m)
    |   movel([0.092240, -1.407487, -2.555056, -0.749847, 1.570796, 1.663036],accel_mss,speed_ms,0,blend_radius_m)
    |   movel([0.092394, -1.407218, -2.555255, -0.749916, 1.570796, 1.663190],accel_mss,speed_ms,0,blend_radius_m)
    |   movel([0.092628, -1.406997, -2.555420, -0.749972, 1.570796, 1.663424],accel_mss,speed_ms,0,blend_radius_m)
    |   movel([0.093075, -1.406771, -2.555588, -0.750030, 1.570796, 1.663871],accel_mss,speed_ms,0,blend_radius_m)
    |   movel([0.095058, -1.406170, -2.556034, -0.750185, 1.570796, 1.665854],accel_mss,speed_ms,0,blend_radius_m)
    |   speed_ms = 0.003
    |   movel([0.095058, -1.393374, -2.550187, -0.768828, 1.570796, 1.665854],accel_mss,speed_ms,0,blend_radius_m)
    |   speed_ms = 1.000
    |   movel([0.095058, -1.368794, -2.538098, -0.805497, 1.570796, 1.665854],accel_mss,speed_ms,0,blend_radius_m)
    |   movel([0.095035, -1.370360, -2.536997, -0.805032, 1.570796, 1.665831],accel_mss,speed_ms,0,blend_radius_m)
    |   movel([0.095035, -1.394911, -2.549067, -0.768411, 1.570796, 1.665831],accel_mss,speed_ms,0,blend_radius_m)
    |   speed_ms = 0.003
    |   movel([0.095035, -1.404463, -2.553458, -0.754468, 1.570796, 1.665831],accel_mss,speed_ms,0,blend_radius_m)
    |   speed_ms = 0.007
    |   movel([0.096678, -1.404013, -2.553791, -0.754585, 1.570796, 1.667474],accel_mss,speed_ms,0,blend_radius_m)
    |   movel([0.097776, -1.403780, -2.553963, -0.754646, 1.570796, 1.668573],accel_mss,speed_ms,0,blend_radius_m)
    |   movel([0.098503, -1.403710, -2.554016, -0.754664, 1.570796, 1.669299],accel_mss,speed_ms,0,blend_radius_m)
    |   movel([0.098867, -1.403822, -2.553932, -0.754635, 1.570796, 1.669663],accel_mss,speed_ms,0,blend_radius_m)
    |   movel([0.098943, -1.404146, -2.553692, -0.754550, 1.570796, 1.669739],accel_mss,speed_ms,0,blend_radius_m)
    |   movel([0.098660, -1.404518, -2.553417, -0.754454, 1.570796, 1.669456],accel_mss,speed_ms,0,blend_radius_m)
    |   movel([0.098382, -1.404581, -2.553370, -0.754438, 1.570796, 1.669178],accel_mss,speed_ms,0,blend_radius_m)
    |   movel([0.098132, -1.404608, -2.553350, -0.754431, 1.570796, 1.668928],accel_mss,speed_ms,0,blend_radius_m)
    |   movel([0.097854, -1.404624, -2.553339, -0.754426, 1.570796, 1.668651],accel_mss,speed_ms,0,blend_radius_m)
    |   movel([0.096922, -1.404748, -2.553246, -0.754394, 1.570796, 1.667719],accel_mss,speed_ms,0,blend_radius_m)
    |   movel([0.095411, -1.405123, -2.552968, -0.754297, 1.570796, 1.666208],accel_mss,speed_ms,0,blend_radius_m)
    |   movel([0.093895, -1.405570, -2.552637, -0.754182, 1.570796, 1.664692],accel_mss,speed_ms,0,blend_radius_m)
    |   movel([0.092949, -1.405958, -2.552349, -0.754082, 1.570796, 1.663745],accel_mss,speed_ms,0,blend_radius_m)
    |   movel([0.092619, -1.406115, -2.552232, -0.754042, 1.570796, 1.663415],accel_mss,speed_ms,0,blend_radius_m)
    |   movel([0.092226, -1.406242, -2.552137, -0.754009, 1.570796, 1.663023],accel_mss,speed_ms,0,blend_radius_m)
    |   movel([0.092027, -1.406107, -2.552238, -0.754044, 1.570796, 1.662823],accel_mss,speed_ms,0,blend_radius_m)
    |   movel([0.092203, -1.405669, -2.552563, -0.754157, 1.570796, 1.663000],accel_mss,speed_ms,0,blend_radius_m)
    |   movel([0.092457, -1.405414, -2.552753, -0.754222, 1.570796, 1.663253],accel_mss,speed_ms,0,blend_radius_m)
    |   movel([0.092744, -1.405218, -2.552898, -0.754273, 1.570796, 1.663541],accel_mss,speed_ms,0,blend_radius_m)
    |   movel([0.093114, -1.405050, -2.553023, -0.754316, 1.570796, 1.663910],accel_mss,speed_ms,0,blend_radius_m)
    |   movel([0.093718, -1.404848, -2.553172, -0.754368, 1.570796, 1.664514],accel_mss,speed_ms,0,blend_radius_m)
    |   movel([0.095035, -1.404463, -2.553458, -0.754468, 1.570796, 1.665831],accel_mss,speed_ms,0,blend_radius_m)
    |   speed_ms = 0.003
    |   movel([0.095035, -1.407689, -2.554905, -0.749795, 1.570796, 1.665831],accel_mss,speed_ms,0,blend_radius_m)
    |   speed_ms = 0.007
    |   movel([0.096678, -1.407240, -2.555239, -0.749910, 1.570796, 1.667474],accel_mss,speed_ms,0,blend_radius_m)
    |   movel([0.097776, -1.407008, -2.555411, -0.749969, 1.570796, 1.668573],accel_mss,speed_ms,0,blend_radius_m)
    |   movel([0.098503, -1.406938, -2.555464, -0.749987, 1.570796, 1.669299],accel_mss,speed_ms,0,blend_radius_m)
    |   movel([0.098867, -1.407050, -2.555380, -0.749959, 1.570796, 1.669663],accel_mss,speed_ms,0,blend_radius_m)
    |   movel([0.098943, -1.407374, -2.555140, -0.749876, 1.570796, 1.669739],accel_mss,speed_ms,0,blend_radius_m)
    |   movel([0.098660, -1.407744, -2.554864, -0.749781, 1.570796, 1.669456],accel_mss,speed_ms,0,blend_radius_m)
    |   movel([0.098382, -1.407807, -2.554817, -0.749765, 1.570796, 1.669178],accel_mss,speed_ms,0,blend_radius_m)
    |   movel([0.098132, -1.407834, -2.554797, -0.749758, 1.570796, 1.668928],accel_mss,speed_ms,0,blend_radius_m)
    |   movel([0.097854, -1.407850, -2.554785, -0.749754, 1.570796, 1.668651],accel_mss,speed_ms,0,blend_radius_m)
    |   movel([0.096922, -1.407974, -2.554693, -0.749722, 1.570796, 1.667719],accel_mss,speed_ms,0,blend_radius_m)
    |   movel([0.095411, -1.408348, -2.554414, -0.749627, 1.570796, 1.666208],accel_mss,speed_ms,0,blend_radius_m)
    |   movel([0.093895, -1.408794, -2.554082, -0.749514, 1.570796, 1.664692],accel_mss,speed_ms,0,blend_radius_m)
    |   movel([0.092949, -1.409180, -2.553793, -0.749416, 1.570796, 1.663745],accel_mss,speed_ms,0,blend_radius_m)
    |   movel([0.092619, -1.409336, -2.553676, -0.749376, 1.570796, 1.663415],accel_mss,speed_ms,0,blend_radius_m)
    |   movel([0.092226, -1.409464, -2.553581, -0.749344, 1.570796, 1.663023],accel_mss,speed_ms,0,blend_radius_m)
    |   movel([0.092027, -1.409329, -2.553682, -0.749378, 1.570796, 1.662823],accel_mss,speed_ms,0,blend_radius_m)
    |   movel([0.092203, -1.408892, -2.554008, -0.749489, 1.570796, 1.663000],accel_mss,speed_ms,0,blend_radius_m)
    |   movel([0.092457, -1.408637, -2.554198, -0.749553, 1.570796, 1.663253],accel_mss,speed_ms,0,blend_radius_m)
    |   movel([0.092744, -1.408442, -2.554344, -0.749603, 1.570796, 1.663541],accel_mss,speed_ms,0,blend_radius_m)
    |   movel([0.093114, -1.408275, -2.554469, -0.749646, 1.570796, 1.663910],accel_mss,speed_ms,0,blend_radius_m)
    |   movel([0.093718, -1.408074, -2.554618, -0.749697, 1.570796, 1.664514],accel_mss,speed_ms,0,blend_radius_m)
    |   movel([0.095035, -1.407689, -2.554905, -0.749795, 1.570796, 1.665831],accel_mss,speed_ms,0,blend_radius_m)
    |   speed_ms = 0.003
    |   movel([0.095035, -1.394911, -2.549067, -0.768411, 1.570796, 1.665831],accel_mss,speed_ms,0,blend_radius_m)
    |   speed_ms = 1.000
    |   movel([0.095035, -1.370360, -2.536997, -0.805032, 1.570796, 1.665831],accel_mss,speed_ms,0,blend_radius_m)
    |   movel([0.094639, -1.371914, -2.535902, -0.804573, 1.570796, 1.665435],accel_mss,speed_ms,0,blend_radius_m)
    |   movel([0.094639, -1.396436, -2.547952, -0.768001, 1.570796, 1.665435],accel_mss,speed_ms,0,blend_radius_m)
    |   speed_ms = 0.003
    |   movel([0.094639, -1.405976, -2.552335, -0.754078, 1.570796, 1.665435],accel_mss,speed_ms,0,blend_radius_m)
    |   speed_ms = 0.007
    |   movel([0.095700, -1.405698, -2.552542, -0.754149, 1.570796, 1.666496],accel_mss,speed_ms,0,blend_radius_m)
    |   movel([0.097708, -1.405190, -2.552919, -0.754280, 1.570796, 1.668504],accel_mss,speed_ms,0,blend_radius_m)
    |   movel([0.098496, -1.405331, -2.552814, -0.754244, 1.570796, 1.669292],accel_mss,speed_ms,0,blend_radius_m)
    |   movel([0.099084, -1.405493, -2.552694, -0.754202, 1.570796, 1.669880],accel_mss,speed_ms,0,blend_radius_m)
    |   movel([0.099446, -1.405731, -2.552517, -0.754141, 1.570796, 1.670242],accel_mss,speed_ms,0,blend_radius_m)
    |   movel([0.099663, -1.406106, -2.552239, -0.754044, 1.570796, 1.670460],accel_mss,speed_ms,0,blend_radius_m)
    |   movel([0.099786, -1.406703, -2.551795, -0.753891, 1.570796, 1.670583],accel_mss,speed_ms,0,blend_radius_m)
    |   movel([0.099688, -1.407004, -2.551571, -0.753814, 1.570796, 1.670484],accel_mss,speed_ms,0,blend_radius_m)
    |   movel([0.099544, -1.407333, -2.551326, -0.753730, 1.570796, 1.670341],accel_mss,speed_ms,0,blend_radius_m)
    |   movel([0.099344, -1.407622, -2.551110, -0.753657, 1.570796, 1.670140],accel_mss,speed_ms,0,blend_radius_m)
    |   movel([0.098360, -1.408089, -2.550762, -0.753538, 1.570796, 1.669156],accel_mss,speed_ms,0,blend_radius_m)
    |   movel([0.096049, -1.408788, -2.550240, -0.753361, 1.570796, 1.666845],accel_mss,speed_ms,0,blend_radius_m)
    |   movel([0.093670, -1.409447, -2.549747, -0.753195, 1.570796, 1.664466],accel_mss,speed_ms,0,blend_radius_m)
    |   movel([0.091851, -1.409859, -2.549439, -0.753091, 1.570796, 1.662647],accel_mss,speed_ms,0,blend_radius_m)
    |   movel([0.091060, -1.409980, -2.549348, -0.753061, 1.570796, 1.661856],accel_mss,speed_ms,0,blend_radius_m)
    |   movel([0.090671, -1.409936, -2.549381, -0.753072, 1.570796, 1.661467],accel_mss,speed_ms,0,blend_radius_m)
    |   movel([0.090493, -1.409731, -2.549535, -0.753123, 1.570796, 1.661289],accel_mss,speed_ms,0,blend_radius_m)
    |   movel([0.090475, -1.409302, -2.549856, -0.753231, 1.570796, 1.661272],accel_mss,speed_ms,0,blend_radius_m)
    |   movel([0.090698, -1.408553, -2.550415, -0.753420, 1.570796, 1.661494],accel_mss,speed_ms,0,blend_radius_m)
    |   movel([0.091185, -1.407836, -2.550951, -0.753602, 1.570796, 1.661982],accel_mss,speed_ms,0,blend_radius_m)
    |   movel([0.091933, -1.407176, -2.551443, -0.753770, 1.570796, 1.662729],accel_mss,speed_ms,0,blend_radius_m)
    |   movel([0.092913, -1.406594, -2.551876, -0.753919, 1.570796, 1.663709],accel_mss,speed_ms,0,blend_radius_m)
    |   movel([0.093405, -1.406375, -2.552039, -0.753975, 1.570796, 1.664201],accel_mss,speed_ms,0,blend_radius_m)
    |   movel([0.093939, -1.406183, -2.552182, -0.754025, 1.570796, 1.664735],accel_mss,speed_ms,0,blend_radius_m)
    |   movel([0.094639, -1.405976, -2.552335, -0.754078, 1.570796, 1.665435],accel_mss,speed_ms,0,blend_radius_m)
    |   speed_ms = 0.003
    |   movel([0.094639, -1.409198, -2.553780, -0.749411, 1.570796, 1.665435],accel_mss,speed_ms,0,blend_radius_m)
    |   speed_ms = 0.007
    |   movel([0.095700, -1.408921, -2.553987, -0.749481, 1.570796, 1.666496],accel_mss,speed_ms,0,blend_radius_m)
    |   movel([0.097708, -1.408414, -2.554365, -0.749610, 1.570796, 1.668504],accel_mss,speed_ms,0,blend_radius_m)
    |   movel([0.098496, -1.408555, -2.554259, -0.749574, 1.570796, 1.669292],accel_mss,speed_ms,0,blend_radius_m)
    |   movel([0.099084, -1.408716, -2.554139, -0.749533, 1.570796, 1.669880],accel_mss,speed_ms,0,blend_radius_m)
    |   movel([0.099446, -1.408954, -2.553962, -0.749473, 1.570796, 1.670242],accel_mss,speed_ms,0,blend_radius_m)
    |   movel([0.099663, -1.409327, -2.553683, -0.749379, 1.570796, 1.670460],accel_mss,speed_ms,0,blend_radius_m)
    |   movel([0.099786, -1.409923, -2.553238, -0.749228, 1.570796, 1.670583],accel_mss,speed_ms,0,blend_radius_m)
    |   movel([0.099688, -1.410223, -2.553014, -0.749152, 1.570796, 1.670484],accel_mss,speed_ms,0,blend_radius_m)
    |   movel([0.099544, -1.410551, -2.552768, -0.749070, 1.570796, 1.670341],accel_mss,speed_ms,0,blend_radius_m)
    |   movel([0.099344, -1.410840, -2.552552, -0.748998, 1.570796, 1.670140],accel_mss,speed_ms,0,blend_radius_m)
    |   movel([0.098360, -1.411305, -2.552203, -0.748881, 1.570796, 1.669156],accel_mss,speed_ms,0,blend_radius_m)
    |   movel([0.096049, -1.412002, -2.551680, -0.748707, 1.570796, 1.666845],accel_mss,speed_ms,0,blend_radius_m)
    |   movel([0.093670, -1.412659, -2.551186, -0.748544, 1.570796, 1.664466],accel_mss,speed_ms,0,blend_radius_m)
    |   movel([0.091851, -1.413070, -2.550877, -0.748442, 1.570796, 1.662647],accel_mss,speed_ms,0,blend_radius_m)
    |   movel([0.091060, -1.413191, -2.550786, -0.748412, 1.570796, 1.661856],accel_mss,speed_ms,0,blend_radius_m)
    |   movel([0.090671, -1.413147, -2.550820, -0.748423, 1.570796, 1.661467],accel_mss,speed_ms,0,blend_radius_m)
    |   movel([0.090493, -1.412943, -2.550973, -0.748473, 1.570796, 1.661289],accel_mss,speed_ms,0,blend_radius_m)
    |   movel([0.090475, -1.412515, -2.551295, -0.748579, 1.570796, 1.661272],accel_mss,speed_ms,0,blend_radius_m)
    |   movel([0.090698, -1.411768, -2.551856, -0.748765, 1.570796, 1.661494],accel_mss,speed_ms,0,blend_radius_m)
    |   movel([0.091185, -1.411053, -2.552392, -0.748944, 1.570796, 1.661982],accel_mss,speed_ms,0,blend_radius_m)
    |   movel([0.091933, -1.410395, -2.552885, -0.749109, 1.570796, 1.662729],accel_mss,speed_ms,0,blend_radius_m)
    |   movel([0.092913, -1.409814, -2.553319, -0.749256, 1.570796, 1.663709],accel_mss,speed_ms,0,blend_radius_m)
    |   movel([0.093405, -1.409596, -2.553483, -0.749311, 1.570796, 1.664201],accel_mss,speed_ms,0,blend_radius_m)
    |   movel([0.093939, -1.409404, -2.553626, -0.749359, 1.570796, 1.664735],accel_mss,speed_ms,0,blend_radius_m)
    |   movel([0.094639, -1.409198, -2.553780, -0.749411, 1.570796, 1.665435],accel_mss,speed_ms,0,blend_radius_m)
    |   speed_ms = 0.003
    |   movel([0.094639, -1.396436, -2.547952, -0.768001, 1.570796, 1.665435],accel_mss,speed_ms,0,blend_radius_m)
    |   speed_ms = 1.000
    |   movel([0.094639, -1.371914, -2.535902, -0.804573, 1.570796, 1.665435],accel_mss,speed_ms,0,blend_radius_m)
    |   movel([0.105149, -1.357142, -2.546182, -0.809066, 1.570796, 1.675945],accel_mss,speed_ms,0,blend_radius_m)
    |   movel([0.105149, -1.381936, -2.558418, -0.772035, 1.570796, 1.675945],accel_mss,speed_ms,0,blend_radius_m)
    |   speed_ms = 0.003
    |   movel([0.105149, -1.391592, -2.562871, -0.757926, 1.570796, 1.675945],accel_mss,speed_ms,0,blend_radius_m)
    |   speed_ms = 0.007
    |   movel([0.104563, -1.391094, -2.563231, -0.758064, 1.570796, 1.675360],accel_mss,speed_ms,0,blend_radius_m)
    |   movel([0.104458, -1.390234, -2.563850, -0.758305, 1.570796, 1.675254],accel_mss,speed_ms,0,blend_radius_m)
    |   movel([0.104866, -1.389249, -2.564559, -0.758581, 1.570796, 1.675663],accel_mss,speed_ms,0,blend_radius_m)
    |   movel([0.105135, -1.388888, -2.564818, -0.758683, 1.570796, 1.675931],accel_mss,speed_ms,0,blend_radius_m)
    |   movel([0.105367, -1.388728, -2.564933, -0.758728, 1.570796, 1.676164],accel_mss,speed_ms,0,blend_radius_m)
    |   movel([0.105422, -1.389121, -2.564651, -0.758617, 1.570796, 1.676219],accel_mss,speed_ms,0,blend_radius_m)
    |   movel([0.105424, -1.389397, -2.564452, -0.758539, 1.570796, 1.676221],accel_mss,speed_ms,0,blend_radius_m)
    |   movel([0.105462, -1.390010, -2.564012, -0.758367, 1.570796, 1.676258],accel_mss,speed_ms,0,blend_radius_m)
    |   movel([0.105618, -1.390484, -2.563670, -0.758235, 1.570796, 1.676415],accel_mss,speed_ms,0,blend_radius_m)
    |   movel([0.105896, -1.390824, -2.563425, -0.758140, 1.570796, 1.676693],accel_mss,speed_ms,0,blend_radius_m)
    |   movel([0.106295, -1.391039, -2.563270, -0.758080, 1.570796, 1.677091],accel_mss,speed_ms,0,blend_radius_m)
    |   movel([0.106601, -1.391184, -2.563166, -0.758039, 1.570796, 1.677397],accel_mss,speed_ms,0,blend_radius_m)
    |   movel([0.106634, -1.391377, -2.563026, -0.757985, 1.570796, 1.677431],accel_mss,speed_ms,0,blend_radius_m)
    |   movel([0.106282, -1.391530, -2.562916, -0.757943, 1.570796, 1.677078],accel_mss,speed_ms,0,blend_radius_m)
    |   movel([0.105149, -1.391592, -2.562871, -0.757926, 1.570796, 1.675945],accel_mss,speed_ms,0,blend_radius_m)
    |   speed_ms = 0.003
    |   movel([0.105149, -1.394854, -2.564339, -0.753196, 1.570796, 1.675945],accel_mss,speed_ms,0,blend_radius_m)
    |   speed_ms = 0.007
    |   movel([0.104563, -1.394357, -2.564699, -0.753332, 1.570796, 1.675360],accel_mss,speed_ms,0,blend_radius_m)
    |   movel([0.104458, -1.393500, -2.565320, -0.753569, 1.570796, 1.675254],accel_mss,speed_ms,0,blend_radius_m)
    |   movel([0.104866, -1.392517, -2.566031, -0.753841, 1.570796, 1.675663],accel_mss,speed_ms,0,blend_radius_m)
    |   movel([0.105135, -1.392158, -2.566290, -0.753941, 1.570796, 1.675931],accel_mss,speed_ms,0,blend_radius_m)
    |   movel([0.105367, -1.391998, -2.566406, -0.753986, 1.570796, 1.676164],accel_mss,speed_ms,0,blend_radius_m)
    |   movel([0.105422, -1.392390, -2.566123, -0.753877, 1.570796, 1.676219],accel_mss,speed_ms,0,blend_radius_m)
    |   movel([0.105424, -1.392666, -2.565923, -0.753800, 1.570796, 1.676221],accel_mss,speed_ms,0,blend_radius_m)
    |   movel([0.105462, -1.393277, -2.565482, -0.753631, 1.570796, 1.676258],accel_mss,speed_ms,0,blend_radius_m)
    |   movel([0.105618, -1.393750, -2.565140, -0.753500, 1.570796, 1.676415],accel_mss,speed_ms,0,blend_radius_m)
    |   movel([0.105896, -1.394089, -2.564894, -0.753406, 1.570796, 1.676693],accel_mss,speed_ms,0,blend_radius_m)
    |   movel([0.106295, -1.394303, -2.564739, -0.753347, 1.570796, 1.677091],accel_mss,speed_ms,0,blend_radius_m)
    |   movel([0.106601, -1.394447, -2.564634, -0.753308, 1.570796, 1.677397],accel_mss,speed_ms,0,blend_radius_m)
    |   movel([0.106634, -1.394640, -2.564494, -0.753255, 1.570796, 1.677431],accel_mss,speed_ms,0,blend_radius_m)
    |   movel([0.106282, -1.394792, -2.564384, -0.753213, 1.570796, 1.677078],accel_mss,speed_ms,0,blend_radius_m)
    |   movel([0.105149, -1.394854, -2.564339, -0.753196, 1.570796, 1.675945],accel_mss,speed_ms,0,blend_radius_m)
    |   speed_ms = 0.003
    |   movel([0.105149, -1.381936, -2.558418, -0.772035, 1.570796, 1.675945],accel_mss,speed_ms,0,blend_radius_m)
    |   speed_ms = 1.000
    |   movel([0.105149, -1.357142, -2.546182, -0.809066, 1.570796, 1.675945],accel_mss,speed_ms,0,blend_radius_m)
    |   movel([0.110232, -1.354325, -2.548108, -0.809956, 1.570796, 1.681029],accel_mss,speed_ms,0,blend_radius_m)
    |   movel([0.110232, -1.379170, -2.560380, -0.772838, 1.570796, 1.681029],accel_mss,speed_ms,0,blend_radius_m)
    |   speed_ms = 0.003
    |   movel([0.110232, -1.388848, -2.564847, -0.758694, 1.570796, 1.681029],accel_mss,speed_ms,0,blend_radius_m)
    |   speed_ms = 0.007
    |   movel([0.110305, -1.388373, -2.565188, -0.758828, 1.570796, 1.681101],accel_mss,speed_ms,0,blend_radius_m)
    |   movel([0.110347, -1.387801, -2.565598, -0.758990, 1.570796, 1.681143],accel_mss,speed_ms,0,blend_radius_m)
    |   movel([0.110245, -1.387322, -2.565941, -0.759126, 1.570796, 1.681042],accel_mss,speed_ms,0,blend_radius_m)
    |   movel([0.109999, -1.386943, -2.566212, -0.759234, 1.570796, 1.680796],accel_mss,speed_ms,0,blend_radius_m)
    |   movel([0.109609, -1.386664, -2.566412, -0.759314, 1.570796, 1.680405],accel_mss,speed_ms,0,blend_radius_m)
    |   movel([0.109341, -1.386511, -2.566521, -0.759357, 1.570796, 1.680137],accel_mss,speed_ms,0,blend_radius_m)
    |   movel([0.109697, -1.386266, -2.566696, -0.759427, 1.570796, 1.680494],accel_mss,speed_ms,0,blend_radius_m)
    |   movel([0.110064, -1.386321, -2.566656, -0.759411, 1.570796, 1.680860],accel_mss,speed_ms,0,blend_radius_m)
    |   movel([0.110479, -1.386543, -2.566498, -0.759348, 1.570796, 1.681275],accel_mss,speed_ms,0,blend_radius_m)
    |   movel([0.110833, -1.386845, -2.566282, -0.759262, 1.570796, 1.681629],accel_mss,speed_ms,0,blend_radius_m)
    |   movel([0.111019, -1.387167, -2.566052, -0.759170, 1.570796, 1.681815],accel_mss,speed_ms,0,blend_radius_m)
    |   movel([0.111077, -1.387536, -2.565788, -0.759065, 1.570796, 1.681873],accel_mss,speed_ms,0,blend_radius_m)
    |   movel([0.111027, -1.387962, -2.565482, -0.758945, 1.570796, 1.681823],accel_mss,speed_ms,0,blend_radius_m)
    |   movel([0.110881, -1.388389, -2.565176, -0.758824, 1.570796, 1.681677],accel_mss,speed_ms,0,blend_radius_m)
    |   movel([0.110658, -1.388753, -2.564915, -0.758721, 1.570796, 1.681454],accel_mss,speed_ms,0,blend_radius_m)
    |   movel([0.110420, -1.389003, -2.564736, -0.758650, 1.570796, 1.681217],accel_mss,speed_ms,0,blend_radius_m)
    |   movel([0.110232, -1.388848, -2.564847, -0.758694, 1.570796, 1.681029],accel_mss,speed_ms,0,blend_radius_m)
    |   speed_ms = 0.003
    |   movel([0.110232, -1.392118, -2.566319, -0.753952, 1.570796, 1.681029],accel_mss,speed_ms,0,blend_radius_m)
    |   speed_ms = 0.007
    |   movel([0.110305, -1.391644, -2.566661, -0.754084, 1.570796, 1.681101],accel_mss,speed_ms,0,blend_radius_m)
    |   movel([0.110347, -1.391074, -2.567071, -0.754244, 1.570796, 1.681143],accel_mss,speed_ms,0,blend_radius_m)
    |   movel([0.110245, -1.390596, -2.567416, -0.754378, 1.570796, 1.681042],accel_mss,speed_ms,0,blend_radius_m)
    |   movel([0.109999, -1.390218, -2.567687, -0.754484, 1.570796, 1.680796],accel_mss,speed_ms,0,blend_radius_m)
    |   movel([0.109609, -1.389940, -2.567887, -0.754562, 1.570796, 1.680405],accel_mss,speed_ms,0,blend_radius_m)
    |   movel([0.109341, -1.389788, -2.567997, -0.754605, 1.570796, 1.680137],accel_mss,speed_ms,0,blend_radius_m)
    |   movel([0.109697, -1.389543, -2.568172, -0.754674, 1.570796, 1.680494],accel_mss,speed_ms,0,blend_radius_m)
    |   movel([0.110064, -1.389598, -2.568133, -0.754658, 1.570796, 1.680860],accel_mss,speed_ms,0,blend_radius_m)
    |   movel([0.110479, -1.389819, -2.567974, -0.754596, 1.570796, 1.681275],accel_mss,speed_ms,0,blend_radius_m)
    |   movel([0.110833, -1.390120, -2.567758, -0.754511, 1.570796, 1.681629],accel_mss,speed_ms,0,blend_radius_m)
    |   movel([0.111019, -1.390441, -2.567527, -0.754421, 1.570796, 1.681815],accel_mss,speed_ms,0,blend_radius_m)
    |   movel([0.111077, -1.390809, -2.567262, -0.754318, 1.570796, 1.681873],accel_mss,speed_ms,0,blend_radius_m)
    |   movel([0.111027, -1.391234, -2.566956, -0.754199, 1.570796, 1.681823],accel_mss,speed_ms,0,blend_radius_m)
    |   movel([0.110881, -1.391660, -2.566649, -0.754080, 1.570796, 1.681677],accel_mss,speed_ms,0,blend_radius_m)
    |   movel([0.110658, -1.392023, -2.566387, -0.753979, 1.570796, 1.681454],accel_mss,speed_ms,0,blend_radius_m)
    |   movel([0.110420, -1.392272, -2.566208, -0.753909, 1.570796, 1.681217],accel_mss,speed_ms,0,blend_radius_m)
    |   movel([0.110232, -1.392118, -2.566319, -0.753952, 1.570796, 1.681029],accel_mss,speed_ms,0,blend_radius_m)
    |   speed_ms = 0.003
    |   movel([0.110232, -1.379170, -2.560380, -0.772838, 1.570796, 1.681029],accel_mss,speed_ms,0,blend_radius_m)
    |   speed_ms = 1.000
    |   movel([0.110232, -1.354325, -2.548108, -0.809956, 1.570796, 1.681029],accel_mss,speed_ms,0,blend_radius_m)
    |   movel([0.107803, -1.351830, -2.549806, -0.810754, 1.570796, 1.678599],accel_mss,speed_ms,0,blend_radius_m)
    |   movel([0.107803, -1.376720, -2.562109, -0.773559, 1.570796, 1.678599],accel_mss,speed_ms,0,blend_radius_m)
    |   speed_ms = 0.003
    |   movel([0.107803, -1.386417, -2.566588, -0.759384, 1.570796, 1.678599],accel_mss,speed_ms,0,blend_radius_m)
    |   speed_ms = 0.007
    |   movel([0.107128, -1.386811, -2.566306, -0.759272, 1.570796, 1.677924],accel_mss,speed_ms,0,blend_radius_m)
    |   movel([0.106731, -1.386981, -2.566185, -0.759223, 1.570796, 1.677527],accel_mss,speed_ms,0,blend_radius_m)
    |   movel([0.106421, -1.387067, -2.566123, -0.759199, 1.570796, 1.677217],accel_mss,speed_ms,0,blend_radius_m)
    |   movel([0.106109, -1.386952, -2.566205, -0.759231, 1.570796, 1.676905],accel_mss,speed_ms,0,blend_radius_m)
    |   movel([0.106253, -1.386718, -2.566373, -0.759298, 1.570796, 1.677049],accel_mss,speed_ms,0,blend_radius_m)
    |   movel([0.106611, -1.386494, -2.566533, -0.759362, 1.570796, 1.677408],accel_mss,speed_ms,0,blend_radius_m)
    |   movel([0.107012, -1.386281, -2.566685, -0.759423, 1.570796, 1.677808],accel_mss,speed_ms,0,blend_radius_m)
    |   movel([0.107410, -1.386119, -2.566801, -0.759469, 1.570796, 1.678207],accel_mss,speed_ms,0,blend_radius_m)
    |   movel([0.107741, -1.386026, -2.566867, -0.759496, 1.570796, 1.678537],accel_mss,speed_ms,0,blend_radius_m)
    |   movel([0.107964, -1.386144, -2.566783, -0.759462, 1.570796, 1.678760],accel_mss,speed_ms,0,blend_radius_m)
    |   movel([0.107803, -1.386417, -2.566588, -0.759384, 1.570796, 1.678599],accel_mss,speed_ms,0,blend_radius_m)
    |   speed_ms = 0.003
    |   movel([0.107803, -1.389693, -2.568064, -0.754631, 1.570796, 1.678599],accel_mss,speed_ms,0,blend_radius_m)
    |   speed_ms = 0.007
    |   movel([0.107128, -1.390086, -2.567782, -0.754521, 1.570796, 1.677924],accel_mss,speed_ms,0,blend_radius_m)
    |   movel([0.106731, -1.390256, -2.567660, -0.754473, 1.570796, 1.677527],accel_mss,speed_ms,0,blend_radius_m)
    |   movel([0.106421, -1.390342, -2.567598, -0.754449, 1.570796, 1.677217],accel_mss,speed_ms,0,blend_radius_m)
    |   movel([0.106109, -1.390227, -2.567681, -0.754481, 1.570796, 1.676905],accel_mss,speed_ms,0,blend_radius_m)
    |   movel([0.106253, -1.389994, -2.567849, -0.754547, 1.570796, 1.677049],accel_mss,speed_ms,0,blend_radius_m)
    |   movel([0.106611, -1.389770, -2.568009, -0.754610, 1.570796, 1.677408],accel_mss,speed_ms,0,blend_radius_m)
    |   movel([0.107012, -1.389558, -2.568161, -0.754669, 1.570796, 1.677808],accel_mss,speed_ms,0,blend_radius_m)
    |   movel([0.107410, -1.389397, -2.568277, -0.754715, 1.570796, 1.678207],accel_mss,speed_ms,0,blend_radius_m)
    |   movel([0.107741, -1.389303, -2.568344, -0.754741, 1.570796, 1.678537],accel_mss,speed_ms,0,blend_radius_m)
    |   movel([0.107964, -1.389422, -2.568259, -0.754708, 1.570796, 1.678760],accel_mss,speed_ms,0,blend_radius_m)
    |   movel([0.107803, -1.389693, -2.568064, -0.754631, 1.570796, 1.678599],accel_mss,speed_ms,0,blend_radius_m)
    |   speed_ms = 0.003
    |   movel([0.107803, -1.376720, -2.562109, -0.773559, 1.570796, 1.678599],accel_mss,speed_ms,0,blend_radius_m)
    |   speed_ms = 1.000
    |   movel([0.107803, -1.351830, -2.549806, -0.810754, 1.570796, 1.678599],accel_mss,speed_ms,0,blend_radius_m)
    |   movel([0.107973, -1.350503, -2.550705, -0.811181, 1.570796, 1.678770],accel_mss,speed_ms,0,blend_radius_m)
    |   movel([0.107973, -1.375417, -2.563025, -0.773946, 1.570796, 1.678770],accel_mss,speed_ms,0,blend_radius_m)
    |   speed_ms = 0.003
    |   movel([0.107973, -1.385124, -2.567510, -0.759754, 1.570796, 1.678770],accel_mss,speed_ms,0,blend_radius_m)
    |   speed_ms = 0.007
    |   movel([0.107603, -1.385250, -2.567421, -0.759718, 1.570796, 1.678399],accel_mss,speed_ms,0,blend_radius_m)
    |   movel([0.107189, -1.385395, -2.567317, -0.759676, 1.570796, 1.677985],accel_mss,speed_ms,0,blend_radius_m)
    |   movel([0.106724, -1.385579, -2.567186, -0.759624, 1.570796, 1.677521],accel_mss,speed_ms,0,blend_radius_m)
    |   movel([0.106276, -1.385774, -2.567047, -0.759568, 1.570796, 1.677072],accel_mss,speed_ms,0,blend_radius_m)
    |   movel([0.105926, -1.385946, -2.566924, -0.759519, 1.570796, 1.676722],accel_mss,speed_ms,0,blend_radius_m)
    |   movel([0.105544, -1.386142, -2.566785, -0.759463, 1.570796, 1.676341],accel_mss,speed_ms,0,blend_radius_m)
    |   movel([0.105157, -1.386272, -2.566691, -0.759425, 1.570796, 1.675953],accel_mss,speed_ms,0,blend_radius_m)
    |   movel([0.105004, -1.386071, -2.566835, -0.759483, 1.570796, 1.675800],accel_mss,speed_ms,0,blend_radius_m)
    |   movel([0.105156, -1.385786, -2.567039, -0.759564, 1.570796, 1.675952],accel_mss,speed_ms,0,blend_radius_m)
    |   movel([0.105471, -1.385463, -2.567269, -0.759657, 1.570796, 1.676268],accel_mss,speed_ms,0,blend_radius_m)
    |   movel([0.105874, -1.385190, -2.567463, -0.759735, 1.570796, 1.676671],accel_mss,speed_ms,0,blend_radius_m)
    |   movel([0.106140, -1.385062, -2.567555, -0.759772, 1.570796, 1.676936],accel_mss,speed_ms,0,blend_radius_m)
    |   movel([0.106547, -1.384893, -2.567675, -0.759821, 1.570796, 1.677344],accel_mss,speed_ms,0,blend_radius_m)
    |   movel([0.107006, -1.384720, -2.567798, -0.759871, 1.570796, 1.677802],accel_mss,speed_ms,0,blend_radius_m)
    |   movel([0.107455, -1.384567, -2.567907, -0.759915, 1.570796, 1.678251],accel_mss,speed_ms,0,blend_radius_m)
    |   movel([0.108037, -1.384386, -2.568036, -0.759967, 1.570796, 1.678833],accel_mss,speed_ms,0,blend_radius_m)
    |   movel([0.108361, -1.384309, -2.568091, -0.759989, 1.570796, 1.679158],accel_mss,speed_ms,0,blend_radius_m)
    |   movel([0.108712, -1.384347, -2.568064, -0.759978, 1.570796, 1.679508],accel_mss,speed_ms,0,blend_radius_m)
    |   movel([0.108880, -1.384554, -2.567917, -0.759918, 1.570796, 1.679677],accel_mss,speed_ms,0,blend_radius_m)
    |   movel([0.108710, -1.384798, -2.567743, -0.759848, 1.570796, 1.679507],accel_mss,speed_ms,0,blend_radius_m)
    |   movel([0.108314, -1.384993, -2.567604, -0.759792, 1.570796, 1.679110],accel_mss,speed_ms,0,blend_radius_m)
    |   movel([0.107973, -1.385124, -2.567510, -0.759754, 1.570796, 1.678770],accel_mss,speed_ms,0,blend_radius_m)
    |   speed_ms = 0.003
    |   movel([0.107973, -1.388404, -2.568989, -0.754996, 1.570796, 1.678770],accel_mss,speed_ms,0,blend_radius_m)
    |   speed_ms = 0.007
    |   movel([0.107603, -1.388529, -2.568899, -0.754961, 1.570796, 1.678399],accel_mss,speed_ms,0,blend_radius_m)
    |   movel([0.107189, -1.388675, -2.568795, -0.754919, 1.570796, 1.677985],accel_mss,speed_ms,0,blend_radius_m)
    |   movel([0.106724, -1.388858, -2.568663, -0.754867, 1.570796, 1.677521],accel_mss,speed_ms,0,blend_radius_m)
    |   movel([0.106276, -1.389052, -2.568524, -0.754812, 1.570796, 1.677072],accel_mss,speed_ms,0,blend_radius_m)
    |   movel([0.105926, -1.389224, -2.568401, -0.754764, 1.570796, 1.676722],accel_mss,speed_ms,0,blend_radius_m)
    |   movel([0.105544, -1.389419, -2.568261, -0.754709, 1.570796, 1.676341],accel_mss,speed_ms,0,blend_radius_m)
    |   movel([0.105157, -1.389549, -2.568168, -0.754672, 1.570796, 1.675953],accel_mss,speed_ms,0,blend_radius_m)
    |   movel([0.105004, -1.389348, -2.568312, -0.754729, 1.570796, 1.675800],accel_mss,speed_ms,0,blend_radius_m)
    |   movel([0.105156, -1.389064, -2.568516, -0.754809, 1.570796, 1.675952],accel_mss,speed_ms,0,blend_radius_m)
    |   movel([0.105471, -1.388742, -2.568747, -0.754900, 1.570796, 1.676268],accel_mss,speed_ms,0,blend_radius_m)
    |   movel([0.105874, -1.388470, -2.568941, -0.754977, 1.570796, 1.676671],accel_mss,speed_ms,0,blend_radius_m)
    |   movel([0.106140, -1.388342, -2.569033, -0.755014, 1.570796, 1.676936],accel_mss,speed_ms,0,blend_radius_m)
    |   movel([0.106547, -1.388173, -2.569154, -0.755062, 1.570796, 1.677344],accel_mss,speed_ms,0,blend_radius_m)
    |   movel([0.107006, -1.388001, -2.569277, -0.755111, 1.570796, 1.677802],accel_mss,speed_ms,0,blend_radius_m)
    |   movel([0.107455, -1.387849, -2.569386, -0.755154, 1.570796, 1.678251],accel_mss,speed_ms,0,blend_radius_m)
    |   movel([0.108037, -1.387668, -2.569515, -0.755205, 1.570796, 1.678833],accel_mss,speed_ms,0,blend_radius_m)
    |   movel([0.108361, -1.387591, -2.569571, -0.755227, 1.570796, 1.679158],accel_mss,speed_ms,0,blend_radius_m)
    |   movel([0.108712, -1.387629, -2.569543, -0.755216, 1.570796, 1.679508],accel_mss,speed_ms,0,blend_radius_m)
    |   movel([0.108880, -1.387836, -2.569396, -0.755158, 1.570796, 1.679677],accel_mss,speed_ms,0,blend_radius_m)
    |   movel([0.108710, -1.388079, -2.569222, -0.755088, 1.570796, 1.679507],accel_mss,speed_ms,0,blend_radius_m)
    |   movel([0.108314, -1.388273, -2.569083, -0.755033, 1.570796, 1.679110],accel_mss,speed_ms,0,blend_radius_m)
    |   movel([0.107973, -1.388404, -2.568989, -0.754996, 1.570796, 1.678770],accel_mss,speed_ms,0,blend_radius_m)
    |   speed_ms = 0.003
    |   movel([0.107973, -1.375417, -2.563025, -0.773946, 1.570796, 1.678770],accel_mss,speed_ms,0,blend_radius_m)
    |   speed_ms = 1.000
    |   movel([0.107973, -1.350503, -2.550705, -0.811181, 1.570796, 1.678770],accel_mss,speed_ms,0,blend_radius_m)
    |   movel([0.108036, -1.349102, -2.551652, -0.811635, 1.570796, 1.678832],accel_mss,speed_ms,0,blend_radius_m)
    |   movel([0.108036, -1.374041, -2.563990, -0.774357, 1.570796, 1.678832],accel_mss,speed_ms,0,blend_radius_m)
    |   speed_ms = 0.003
    |   movel([0.108036, -1.383759, -2.568482, -0.760148, 1.570796, 1.678832],accel_mss,speed_ms,0,blend_radius_m)
    |   speed_ms = 0.007
    |   movel([0.107706, -1.383861, -2.568410, -0.760119, 1.570796, 1.678502],accel_mss,speed_ms,0,blend_radius_m)
    |   movel([0.107286, -1.384012, -2.568302, -0.760075, 1.570796, 1.678082],accel_mss,speed_ms,0,blend_radius_m)
    |   movel([0.106844, -1.384185, -2.568179, -0.760025, 1.570796, 1.677640],accel_mss,speed_ms,0,blend_radius_m)
    |   movel([0.106453, -1.384354, -2.568059, -0.759976, 1.570796, 1.677249],accel_mss,speed_ms,0,blend_radius_m)
    |   movel([0.105610, -1.384723, -2.567796, -0.759870, 1.570796, 1.676406],accel_mss,speed_ms,0,blend_radius_m)
    |   movel([0.105148, -1.384885, -2.567681, -0.759823, 1.570796, 1.675944],accel_mss,speed_ms,0,blend_radius_m)
    |   movel([0.104900, -1.384909, -2.567664, -0.759816, 1.570796, 1.675696],accel_mss,speed_ms,0,blend_radius_m)
    |   movel([0.104960, -1.384453, -2.567989, -0.759948, 1.570796, 1.675757],accel_mss,speed_ms,0,blend_radius_m)
    |   movel([0.105494, -1.384038, -2.568284, -0.760067, 1.570796, 1.676290],accel_mss,speed_ms,0,blend_radius_m)
    |   movel([0.106400, -1.383572, -2.568615, -0.760202, 1.570796, 1.677196],accel_mss,speed_ms,0,blend_radius_m)
    |   movel([0.107695, -1.383060, -2.568978, -0.760351, 1.570796, 1.678491],accel_mss,speed_ms,0,blend_radius_m)
    |   movel([0.108125, -1.382914, -2.569082, -0.760393, 1.570796, 1.678921],accel_mss,speed_ms,0,blend_radius_m)
    |   movel([0.108375, -1.382859, -2.569121, -0.760409, 1.570796, 1.679171],accel_mss,speed_ms,0,blend_radius_m)
    |   movel([0.108765, -1.382928, -2.569072, -0.760389, 1.570796, 1.679562],accel_mss,speed_ms,0,blend_radius_m)
    |   movel([0.108980, -1.383039, -2.568993, -0.760357, 1.570796, 1.679776],accel_mss,speed_ms,0,blend_radius_m)
    |   movel([0.109022, -1.383237, -2.568853, -0.760299, 1.570796, 1.679819],accel_mss,speed_ms,0,blend_radius_m)
    |   movel([0.108786, -1.383474, -2.568684, -0.760231, 1.570796, 1.679582],accel_mss,speed_ms,0,blend_radius_m)
    |   movel([0.108311, -1.383674, -2.568543, -0.760173, 1.570796, 1.679107],accel_mss,speed_ms,0,blend_radius_m)
    |   movel([0.108036, -1.383759, -2.568482, -0.760148, 1.570796, 1.678832],accel_mss,speed_ms,0,blend_radius_m)
    |   speed_ms = 0.003
    |   movel([0.108036, -1.387042, -2.569963, -0.755384, 1.570796, 1.678832],accel_mss,speed_ms,0,blend_radius_m)
    |   speed_ms = 0.007
    |   movel([0.107706, -1.387144, -2.569890, -0.755355, 1.570796, 1.678502],accel_mss,speed_ms,0,blend_radius_m)
    |   movel([0.107286, -1.387296, -2.569782, -0.755312, 1.570796, 1.678082],accel_mss,speed_ms,0,blend_radius_m)
    |   movel([0.106844, -1.387467, -2.569659, -0.755263, 1.570796, 1.677640],accel_mss,speed_ms,0,blend_radius_m)
    |   movel([0.106453, -1.387636, -2.569539, -0.755215, 1.570796, 1.677249],accel_mss,speed_ms,0,blend_radius_m)
    |   movel([0.105610, -1.388004, -2.569275, -0.755110, 1.570796, 1.676406],accel_mss,speed_ms,0,blend_radius_m)
    |   movel([0.105148, -1.388165, -2.569160, -0.755064, 1.570796, 1.675944],accel_mss,speed_ms,0,blend_radius_m)
    |   movel([0.104900, -1.388189, -2.569143, -0.755057, 1.570796, 1.675696],accel_mss,speed_ms,0,blend_radius_m)
    |   movel([0.104960, -1.387735, -2.569468, -0.755186, 1.570796, 1.675757],accel_mss,speed_ms,0,blend_radius_m)
    |   movel([0.105494, -1.387321, -2.569764, -0.755304, 1.570796, 1.676290],accel_mss,speed_ms,0,blend_radius_m)
    |   movel([0.106400, -1.386856, -2.570096, -0.755437, 1.570796, 1.677196],accel_mss,speed_ms,0,blend_radius_m)
    |   movel([0.107695, -1.386346, -2.570460, -0.755583, 1.570796, 1.678491],accel_mss,speed_ms,0,blend_radius_m)
    |   movel([0.108125, -1.386200, -2.570564, -0.755625, 1.570796, 1.678921],accel_mss,speed_ms,0,blend_radius_m)
    |   movel([0.108375, -1.386145, -2.570603, -0.755641, 1.570796, 1.679171],accel_mss,speed_ms,0,blend_radius_m)
    |   movel([0.108765, -1.386214, -2.570554, -0.755621, 1.570796, 1.679562],accel_mss,speed_ms,0,blend_radius_m)
    |   movel([0.108980, -1.386325, -2.570475, -0.755589, 1.570796, 1.679776],accel_mss,speed_ms,0,blend_radius_m)
    |   movel([0.109022, -1.386522, -2.570334, -0.755533, 1.570796, 1.679819],accel_mss,speed_ms,0,blend_radius_m)
    |   movel([0.108786, -1.386759, -2.570165, -0.755465, 1.570796, 1.679582],accel_mss,speed_ms,0,blend_radius_m)
    |   movel([0.108311, -1.386958, -2.570023, -0.755408, 1.570796, 1.679107],accel_mss,speed_ms,0,blend_radius_m)
    |   movel([0.108036, -1.387042, -2.569963, -0.755384, 1.570796, 1.678832],accel_mss,speed_ms,0,blend_radius_m)
    |   speed_ms = 0.003
    |   movel([0.108036, -1.374041, -2.563990, -0.774357, 1.570796, 1.678832],accel_mss,speed_ms,0,blend_radius_m)
    |   speed_ms = 1.000
    |   movel([0.108036, -1.349102, -2.551652, -0.811635, 1.570796, 1.678832],accel_mss,speed_ms,0,blend_radius_m)
    |   movel([0.108046, -1.347695, -2.552600, -0.812094, 1.570796, 1.678842],accel_mss,speed_ms,0,blend_radius_m)
    |   movel([0.108046, -1.372660, -2.564956, -0.774773, 1.570796, 1.678842],accel_mss,speed_ms,0,blend_radius_m)
    |   speed_ms = 0.003
    |   movel([0.108046, -1.382388, -2.569455, -0.760546, 1.570796, 1.678842],accel_mss,speed_ms,0,blend_radius_m)
    |   speed_ms = 0.007
    |   movel([0.107493, -1.382574, -2.569323, -0.760492, 1.570796, 1.678290],accel_mss,speed_ms,0,blend_radius_m)
    |   movel([0.106983, -1.382746, -2.569201, -0.760442, 1.570796, 1.677780],accel_mss,speed_ms,0,blend_radius_m)
    |   movel([0.106468, -1.382941, -2.569063, -0.760385, 1.570796, 1.677264],accel_mss,speed_ms,0,blend_radius_m)
    |   movel([0.106014, -1.383128, -2.568930, -0.760331, 1.570796, 1.676811],accel_mss,speed_ms,0,blend_radius_m)
    |   movel([0.105727, -1.383271, -2.568828, -0.760289, 1.570796, 1.676524],accel_mss,speed_ms,0,blend_radius_m)
    |   movel([0.105343, -1.383462, -2.568693, -0.760234, 1.570796, 1.676139],accel_mss,speed_ms,0,blend_radius_m)
    |   movel([0.104988, -1.383409, -2.568731, -0.760249, 1.570796, 1.675785],accel_mss,speed_ms,0,blend_radius_m)
    |   movel([0.104973, -1.383177, -2.568895, -0.760317, 1.570796, 1.675770],accel_mss,speed_ms,0,blend_radius_m)
    |   movel([0.105166, -1.382821, -2.569148, -0.760420, 1.570796, 1.675962],accel_mss,speed_ms,0,blend_radius_m)
    |   movel([0.105621, -1.382469, -2.569397, -0.760522, 1.570796, 1.676417],accel_mss,speed_ms,0,blend_radius_m)
    |   movel([0.106415, -1.382080, -2.569673, -0.760636, 1.570796, 1.677212],accel_mss,speed_ms,0,blend_radius_m)
    |   movel([0.107697, -1.381596, -2.570015, -0.760777, 1.570796, 1.678493],accel_mss,speed_ms,0,blend_radius_m)
    |   movel([0.108165, -1.381440, -2.570126, -0.760823, 1.570796, 1.678961],accel_mss,speed_ms,0,blend_radius_m)
    |   movel([0.108430, -1.381380, -2.570169, -0.760841, 1.570796, 1.679226],accel_mss,speed_ms,0,blend_radius_m)
    |   movel([0.108831, -1.381447, -2.570121, -0.760821, 1.570796, 1.679627],accel_mss,speed_ms,0,blend_radius_m)
    |   movel([0.109048, -1.381564, -2.570039, -0.760787, 1.570796, 1.679844],accel_mss,speed_ms,0,blend_radius_m)
    |   movel([0.109077, -1.381790, -2.569878, -0.760721, 1.570796, 1.679873],accel_mss,speed_ms,0,blend_radius_m)
    |   movel([0.108772, -1.382086, -2.569669, -0.760634, 1.570796, 1.679569],accel_mss,speed_ms,0,blend_radius_m)
    |   movel([0.108466, -1.382226, -2.569570, -0.760593, 1.570796, 1.679262],accel_mss,speed_ms,0,blend_radius_m)
    |   movel([0.108046, -1.382388, -2.569455, -0.760546, 1.570796, 1.678842],accel_mss,speed_ms,0,blend_radius_m)
    |   speed_ms = 0.003
    |   movel([0.108046, -1.385676, -2.570938, -0.755776, 1.570796, 1.678842],accel_mss,speed_ms,0,blend_radius_m)
    |   speed_ms = 0.007
    |   movel([0.107493, -1.385861, -2.570805, -0.755722, 1.570796, 1.678290],accel_mss,speed_ms,0,blend_radius_m)
    |   movel([0.106983, -1.386033, -2.570683, -0.755673, 1.570796, 1.677780],accel_mss,speed_ms,0,blend_radius_m)
    |   movel([0.106468, -1.386227, -2.570544, -0.755617, 1.570796, 1.677264],accel_mss,speed_ms,0,blend_radius_m)
    |   movel([0.106014, -1.386413, -2.570412, -0.755564, 1.570796, 1.676811],accel_mss,speed_ms,0,blend_radius_m)
    |   movel([0.105727, -1.386556, -2.570310, -0.755523, 1.570796, 1.676524],accel_mss,speed_ms,0,blend_radius_m)
    |   movel([0.105343, -1.386746, -2.570174, -0.755469, 1.570796, 1.676139],accel_mss,speed_ms,0,blend_radius_m)
    |   movel([0.104988, -1.386693, -2.570212, -0.755484, 1.570796, 1.675785],accel_mss,speed_ms,0,blend_radius_m)
    |   movel([0.104973, -1.386462, -2.570377, -0.755550, 1.570796, 1.675770],accel_mss,speed_ms,0,blend_radius_m)
    |   movel([0.105166, -1.386108, -2.570630, -0.755652, 1.570796, 1.675962],accel_mss,speed_ms,0,blend_radius_m)
    |   movel([0.105621, -1.385756, -2.570880, -0.755753, 1.570796, 1.676417],accel_mss,speed_ms,0,blend_radius_m)
    |   movel([0.106415, -1.385369, -2.571156, -0.755864, 1.570796, 1.677212],accel_mss,speed_ms,0,blend_radius_m)
    |   movel([0.107697, -1.384886, -2.571499, -0.756003, 1.570796, 1.678493],accel_mss,speed_ms,0,blend_radius_m)
    |   movel([0.108165, -1.384730, -2.571611, -0.756049, 1.570796, 1.678961],accel_mss,speed_ms,0,blend_radius_m)
    |   movel([0.108430, -1.384670, -2.571653, -0.756066, 1.570796, 1.679226],accel_mss,speed_ms,0,blend_radius_m)
    |   movel([0.108831, -1.384737, -2.571606, -0.756047, 1.570796, 1.679627],accel_mss,speed_ms,0,blend_radius_m)
    |   movel([0.109048, -1.384853, -2.571523, -0.756013, 1.570796, 1.679844],accel_mss,speed_ms,0,blend_radius_m)
    |   movel([0.109077, -1.385079, -2.571362, -0.755948, 1.570796, 1.679873],accel_mss,speed_ms,0,blend_radius_m)
    |   movel([0.108772, -1.385374, -2.571152, -0.755863, 1.570796, 1.679569],accel_mss,speed_ms,0,blend_radius_m)
    |   movel([0.108466, -1.385514, -2.571053, -0.755822, 1.570796, 1.679262],accel_mss,speed_ms,0,blend_radius_m)
    |   movel([0.108046, -1.385676, -2.570938, -0.755776, 1.570796, 1.678842],accel_mss,speed_ms,0,blend_radius_m)
    |   speed_ms = 0.003
    |   movel([0.108046, -1.372660, -2.564956, -0.774773, 1.570796, 1.678842],accel_mss,speed_ms,0,blend_radius_m)
    |   speed_ms = 1.000
    |   movel([0.108046, -1.347695, -2.552600, -0.812094, 1.570796, 1.678842],accel_mss,speed_ms,0,blend_radius_m)
    |   movel([0.107957, -1.346153, -2.553637, -0.812600, 1.570796, 1.678753],accel_mss,speed_ms,0,blend_radius_m)
    |   movel([0.107957, -1.371145, -2.566013, -0.775232, 1.570796, 1.678753],accel_mss,speed_ms,0,blend_radius_m)
    |   speed_ms = 0.003
    |   movel([0.107957, -1.380885, -2.570519, -0.760986, 1.570796, 1.678753],accel_mss,speed_ms,0,blend_radius_m)
    |   speed_ms = 0.007
    |   movel([0.107460, -1.381077, -2.570383, -0.760929, 1.570796, 1.678256],accel_mss,speed_ms,0,blend_radius_m)
    |   movel([0.106951, -1.381270, -2.570246, -0.760873, 1.570796, 1.677748],accel_mss,speed_ms,0,blend_radius_m)
    |   movel([0.106468, -1.381455, -2.570116, -0.760819, 1.570796, 1.677264],accel_mss,speed_ms,0,blend_radius_m)
    |   movel([0.106060, -1.381617, -2.570001, -0.760771, 1.570796, 1.676856],accel_mss,speed_ms,0,blend_radius_m)
    |   movel([0.105690, -1.381764, -2.569897, -0.760728, 1.570796, 1.676486],accel_mss,speed_ms,0,blend_radius_m)
    |   movel([0.105469, -1.381660, -2.569971, -0.760759, 1.570796, 1.676265],accel_mss,speed_ms,0,blend_radius_m)
    |   movel([0.105525, -1.381301, -2.570224, -0.760864, 1.570796, 1.676321],accel_mss,speed_ms,0,blend_radius_m)
    |   movel([0.105823, -1.380972, -2.570457, -0.760960, 1.570796, 1.676619],accel_mss,speed_ms,0,blend_radius_m)
    |   movel([0.106443, -1.380643, -2.570689, -0.761057, 1.570796, 1.677239],accel_mss,speed_ms,0,blend_radius_m)
    |   movel([0.107505, -1.380266, -2.570955, -0.761167, 1.570796, 1.678302],accel_mss,speed_ms,0,blend_radius_m)
    |   movel([0.108170, -1.380061, -2.571100, -0.761228, 1.570796, 1.678967],accel_mss,speed_ms,0,blend_radius_m)
    |   movel([0.108524, -1.379975, -2.571160, -0.761253, 1.570796, 1.679320],accel_mss,speed_ms,0,blend_radius_m)
    |   movel([0.108896, -1.380010, -2.571136, -0.761243, 1.570796, 1.679692],accel_mss,speed_ms,0,blend_radius_m)
    |   movel([0.109065, -1.380218, -2.570989, -0.761182, 1.570796, 1.679862],accel_mss,speed_ms,0,blend_radius_m)
    |   movel([0.108895, -1.380457, -2.570821, -0.761111, 1.570796, 1.679692],accel_mss,speed_ms,0,blend_radius_m)
    |   movel([0.108402, -1.380701, -2.570649, -0.761040, 1.570796, 1.679198],accel_mss,speed_ms,0,blend_radius_m)
    |   movel([0.107957, -1.380885, -2.570519, -0.760986, 1.570796, 1.678753],accel_mss,speed_ms,0,blend_radius_m)
    |   speed_ms = 0.003
    |   movel([0.107957, -1.384176, -2.572004, -0.756209, 1.570796, 1.678753],accel_mss,speed_ms,0,blend_radius_m)
    |   speed_ms = 0.007
    |   movel([0.107460, -1.384368, -2.571868, -0.756153, 1.570796, 1.678256],accel_mss,speed_ms,0,blend_radius_m)
    |   movel([0.106951, -1.384561, -2.571731, -0.756097, 1.570796, 1.677748],accel_mss,speed_ms,0,blend_radius_m)
    |   movel([0.106468, -1.384745, -2.571600, -0.756044, 1.570796, 1.677264],accel_mss,speed_ms,0,blend_radius_m)
    |   movel([0.106060, -1.384907, -2.571485, -0.755998, 1.570796, 1.676856],accel_mss,speed_ms,0,blend_radius_m)
    |   movel([0.105690, -1.385054, -2.571380, -0.755955, 1.570796, 1.676486],accel_mss,speed_ms,0,blend_radius_m)
    |   movel([0.105469, -1.384949, -2.571454, -0.755985, 1.570796, 1.676265],accel_mss,speed_ms,0,blend_radius_m)
    |   movel([0.105525, -1.384592, -2.571709, -0.756089, 1.570796, 1.676321],accel_mss,speed_ms,0,blend_radius_m)
    |   movel([0.105823, -1.384264, -2.571942, -0.756184, 1.570796, 1.676619],accel_mss,speed_ms,0,blend_radius_m)
    |   movel([0.106443, -1.383935, -2.572175, -0.756279, 1.570796, 1.677239],accel_mss,speed_ms,0,blend_radius_m)
    |   movel([0.107505, -1.383559, -2.572442, -0.756388, 1.570796, 1.678302],accel_mss,speed_ms,0,blend_radius_m)
    |   movel([0.108170, -1.383355, -2.572586, -0.756447, 1.570796, 1.678967],accel_mss,speed_ms,0,blend_radius_m)
    |   movel([0.108524, -1.383269, -2.572647, -0.756472, 1.570796, 1.679320],accel_mss,speed_ms,0,blend_radius_m)
    |   movel([0.108896, -1.383304, -2.572622, -0.756462, 1.570796, 1.679692],accel_mss,speed_ms,0,blend_radius_m)
    |   movel([0.109065, -1.383511, -2.572476, -0.756402, 1.570796, 1.679862],accel_mss,speed_ms,0,blend_radius_m)
    |   movel([0.108895, -1.383750, -2.572306, -0.756333, 1.570796, 1.679692],accel_mss,speed_ms,0,blend_radius_m)
    |   movel([0.108402, -1.383993, -2.572134, -0.756262, 1.570796, 1.679198],accel_mss,speed_ms,0,blend_radius_m)
    |   movel([0.107957, -1.384176, -2.572004, -0.756209, 1.570796, 1.678753],accel_mss,speed_ms,0,blend_radius_m)
    |   speed_ms = 0.003
    |   movel([0.107957, -1.371145, -2.566013, -0.775232, 1.570796, 1.678753],accel_mss,speed_ms,0,blend_radius_m)
    |   speed_ms = 1.000
    |   movel([0.107957, -1.346153, -2.553637, -0.812600, 1.570796, 1.678753],accel_mss,speed_ms,0,blend_radius_m)
    |   movel([0.107938, -1.344656, -2.554639, -0.813093, 1.570796, 1.678735],accel_mss,speed_ms,0,blend_radius_m)
    |   movel([0.107938, -1.369675, -2.567035, -0.775680, 1.570796, 1.678735],accel_mss,speed_ms,0,blend_radius_m)
    |   speed_ms = 0.003
    |   movel([0.107938, -1.379426, -2.571548, -0.761415, 1.570796, 1.678735],accel_mss,speed_ms,0,blend_radius_m)
    |   speed_ms = 0.007
    |   movel([0.107342, -1.379621, -2.571410, -0.761358, 1.570796, 1.678138],accel_mss,speed_ms,0,blend_radius_m)
    |   movel([0.107347, -1.379363, -2.571592, -0.761434, 1.570796, 1.678143],accel_mss,speed_ms,0,blend_radius_m)
    |   movel([0.107964, -1.378932, -2.571896, -0.761562, 1.570796, 1.678760],accel_mss,speed_ms,0,blend_radius_m)
    |   movel([0.108387, -1.378656, -2.572089, -0.761643, 1.570796, 1.679184],accel_mss,speed_ms,0,blend_radius_m)
    |   movel([0.108732, -1.378526, -2.572181, -0.761682, 1.570796, 1.679529],accel_mss,speed_ms,0,blend_radius_m)
    |   movel([0.108975, -1.378670, -2.572080, -0.761639, 1.570796, 1.679772],accel_mss,speed_ms,0,blend_radius_m)
    |   movel([0.108836, -1.379009, -2.571842, -0.761539, 1.570796, 1.679632],accel_mss,speed_ms,0,blend_radius_m)
    |   movel([0.108501, -1.379192, -2.571712, -0.761484, 1.570796, 1.679298],accel_mss,speed_ms,0,blend_radius_m)
    |   movel([0.108228, -1.379313, -2.571627, -0.761449, 1.570796, 1.679024],accel_mss,speed_ms,0,blend_radius_m)
    |   movel([0.107938, -1.379426, -2.571548, -0.761415, 1.570796, 1.678735],accel_mss,speed_ms,0,blend_radius_m)
    |   speed_ms = 0.003
    |   movel([0.107938, -1.382722, -2.573035, -0.756632, 1.570796, 1.678735],accel_mss,speed_ms,0,blend_radius_m)
    |   speed_ms = 0.007
    |   movel([0.107342, -1.382916, -2.572898, -0.756575, 1.570796, 1.678138],accel_mss,speed_ms,0,blend_radius_m)
    |   movel([0.107347, -1.382659, -2.573079, -0.756650, 1.570796, 1.678143],accel_mss,speed_ms,0,blend_radius_m)
    |   movel([0.107964, -1.382229, -2.573384, -0.756776, 1.570796, 1.678760],accel_mss,speed_ms,0,blend_radius_m)
    |   movel([0.108387, -1.381954, -2.573578, -0.756857, 1.570796, 1.679184],accel_mss,speed_ms,0,blend_radius_m)
    |   movel([0.108732, -1.381824, -2.573670, -0.756895, 1.570796, 1.679529],accel_mss,speed_ms,0,blend_radius_m)
    |   movel([0.108975, -1.381968, -2.573569, -0.756853, 1.570796, 1.679772],accel_mss,speed_ms,0,blend_radius_m)
    |   movel([0.108836, -1.382305, -2.573330, -0.756754, 1.570796, 1.679632],accel_mss,speed_ms,0,blend_radius_m)
    |   movel([0.108501, -1.382489, -2.573200, -0.756700, 1.570796, 1.679298],accel_mss,speed_ms,0,blend_radius_m)
    |   movel([0.108228, -1.382609, -2.573115, -0.756665, 1.570796, 1.679024],accel_mss,speed_ms,0,blend_radius_m)
    |   movel([0.107938, -1.382722, -2.573035, -0.756632, 1.570796, 1.678735],accel_mss,speed_ms,0,blend_radius_m)
    |   speed_ms = 0.003
    |   movel([0.107938, -1.369675, -2.567035, -0.775680, 1.570796, 1.678735],accel_mss,speed_ms,0,blend_radius_m)
    |   speed_ms = 1.000
    |   movel([0.107938, -1.344656, -2.554639, -0.813093, 1.570796, 1.678735],accel_mss,speed_ms,0,blend_radius_m)
    |   movel([0.107459, -1.343867, -2.555167, -0.813355, 1.570796, 1.678255],accel_mss,speed_ms,0,blend_radius_m)
    |   movel([0.107459, -1.368899, -2.567572, -0.775917, 1.570796, 1.678255],accel_mss,speed_ms,0,blend_radius_m)
    |   speed_ms = 0.003
    |   movel([0.107459, -1.378656, -2.572089, -0.761643, 1.570796, 1.678255],accel_mss,speed_ms,0,blend_radius_m)
    |   speed_ms = 0.007
    |   movel([0.106787, -1.379080, -2.571791, -0.761518, 1.570796, 1.677584],accel_mss,speed_ms,0,blend_radius_m)
    |   movel([0.106338, -1.379277, -2.571652, -0.761459, 1.570796, 1.677134],accel_mss,speed_ms,0,blend_radius_m)
    |   movel([0.106106, -1.379255, -2.571668, -0.761466, 1.570796, 1.676902],accel_mss,speed_ms,0,blend_radius_m)
    |   movel([0.106047, -1.379065, -2.571802, -0.761522, 1.570796, 1.676843],accel_mss,speed_ms,0,blend_radius_m)
    |   movel([0.106228, -1.377942, -2.572592, -0.761856, 1.570796, 1.677025],accel_mss,speed_ms,0,blend_radius_m)
    |   movel([0.106395, -1.376860, -2.573350, -0.762179, 1.570796, 1.677191],accel_mss,speed_ms,0,blend_radius_m)
    |   movel([0.106578, -1.375631, -2.574211, -0.762547, 1.570796, 1.677374],accel_mss,speed_ms,0,blend_radius_m)
    |   movel([0.106821, -1.374030, -2.575328, -0.763031, 1.570796, 1.677617],accel_mss,speed_ms,0,blend_radius_m)
    |   movel([0.106988, -1.373093, -2.575980, -0.763316, 1.570796, 1.677784],accel_mss,speed_ms,0,blend_radius_m)
    |   movel([0.107121, -1.372467, -2.576415, -0.763507, 1.570796, 1.677917],accel_mss,speed_ms,0,blend_radius_m)
    |   movel([0.107666, -1.372082, -2.576682, -0.763625, 1.570796, 1.678462],accel_mss,speed_ms,0,blend_radius_m)
    |   movel([0.108309, -1.372101, -2.576669, -0.763619, 1.570796, 1.679105],accel_mss,speed_ms,0,blend_radius_m)
    |   movel([0.108956, -1.372304, -2.576528, -0.763557, 1.570796, 1.679752],accel_mss,speed_ms,0,blend_radius_m)
    |   movel([0.109432, -1.372658, -2.576282, -0.763449, 1.570796, 1.680228],accel_mss,speed_ms,0,blend_radius_m)
    |   movel([0.109711, -1.373202, -2.575904, -0.763283, 1.570796, 1.680507],accel_mss,speed_ms,0,blend_radius_m)
    |   movel([0.109808, -1.374012, -2.575341, -0.763037, 1.570796, 1.680604],accel_mss,speed_ms,0,blend_radius_m)
    |   movel([0.109726, -1.375002, -2.574650, -0.762737, 1.570796, 1.680523],accel_mss,speed_ms,0,blend_radius_m)
    |   movel([0.109459, -1.376100, -2.573883, -0.762407, 1.570796, 1.680255],accel_mss,speed_ms,0,blend_radius_m)
    |   movel([0.109156, -1.376853, -2.573355, -0.762181, 1.570796, 1.679952],accel_mss,speed_ms,0,blend_radius_m)
    |   movel([0.108739, -1.377506, -2.572897, -0.761985, 1.570796, 1.679536],accel_mss,speed_ms,0,blend_radius_m)
    |   movel([0.108184, -1.378094, -2.572485, -0.761810, 1.570796, 1.678981],accel_mss,speed_ms,0,blend_radius_m)
    |   movel([0.107459, -1.378656, -2.572089, -0.761643, 1.570796, 1.678255],accel_mss,speed_ms,0,blend_radius_m)
    |   speed_ms = 0.003
    |   movel([0.107459, -1.381954, -2.573578, -0.756857, 1.570796, 1.678255],accel_mss,speed_ms,0,blend_radius_m)
    |   speed_ms = 0.007
    |   movel([0.106787, -1.382377, -2.573279, -0.756733, 1.570796, 1.677584],accel_mss,speed_ms,0,blend_radius_m)
    |   movel([0.106338, -1.382573, -2.573140, -0.756676, 1.570796, 1.677134],accel_mss,speed_ms,0,blend_radius_m)
    |   movel([0.106106, -1.382551, -2.573156, -0.756682, 1.570796, 1.676902],accel_mss,speed_ms,0,blend_radius_m)
    |   movel([0.106047, -1.382362, -2.573290, -0.756737, 1.570796, 1.676843],accel_mss,speed_ms,0,blend_radius_m)
    |   movel([0.106228, -1.381241, -2.574082, -0.757066, 1.570796, 1.677025],accel_mss,speed_ms,0,blend_radius_m)
    |   movel([0.106395, -1.380163, -2.574842, -0.757384, 1.570796, 1.677191],accel_mss,speed_ms,0,blend_radius_m)
    |   movel([0.106578, -1.378937, -2.575704, -0.757748, 1.570796, 1.677374],accel_mss,speed_ms,0,blend_radius_m)
    |   movel([0.106821, -1.377340, -2.576824, -0.758225, 1.570796, 1.677617],accel_mss,speed_ms,0,blend_radius_m)
    |   movel([0.106988, -1.376405, -2.577478, -0.758505, 1.570796, 1.677784],accel_mss,speed_ms,0,blend_radius_m)
    |   movel([0.107121, -1.375781, -2.577914, -0.758694, 1.570796, 1.677917],accel_mss,speed_ms,0,blend_radius_m)
    |   movel([0.107666, -1.375398, -2.578182, -0.758810, 1.570796, 1.678462],accel_mss,speed_ms,0,blend_radius_m)
    |   movel([0.108309, -1.375417, -2.578168, -0.758804, 1.570796, 1.679105],accel_mss,speed_ms,0,blend_radius_m)
    |   movel([0.108956, -1.375619, -2.578027, -0.758743, 1.570796, 1.679752],accel_mss,speed_ms,0,blend_radius_m)
    |   movel([0.109432, -1.375972, -2.577781, -0.758636, 1.570796, 1.680228],accel_mss,speed_ms,0,blend_radius_m)
    |   movel([0.109711, -1.376515, -2.577402, -0.758473, 1.570796, 1.680507],accel_mss,speed_ms,0,blend_radius_m)
    |   movel([0.109808, -1.377322, -2.576837, -0.758230, 1.570796, 1.680604],accel_mss,speed_ms,0,blend_radius_m)
    |   movel([0.109726, -1.378310, -2.576144, -0.757935, 1.570796, 1.680523],accel_mss,speed_ms,0,blend_radius_m)
    |   movel([0.109459, -1.379404, -2.575376, -0.757609, 1.570796, 1.680255],accel_mss,speed_ms,0,blend_radius_m)
    |   movel([0.109156, -1.380156, -2.574847, -0.757386, 1.570796, 1.679952],accel_mss,speed_ms,0,blend_radius_m)
    |   movel([0.108739, -1.380807, -2.574388, -0.757194, 1.570796, 1.679536],accel_mss,speed_ms,0,blend_radius_m)
    |   movel([0.108184, -1.381393, -2.573975, -0.757021, 1.570796, 1.678981],accel_mss,speed_ms,0,blend_radius_m)
    |   movel([0.107459, -1.381954, -2.573578, -0.756857, 1.570796, 1.678255],accel_mss,speed_ms,0,blend_radius_m)
    |   speed_ms = 0.003
    |   movel([0.107459, -1.368899, -2.567572, -0.775917, 1.570796, 1.678255],accel_mss,speed_ms,0,blend_radius_m)
    |   speed_ms = 1.000
    |   movel([0.107459, -1.343867, -2.555167, -0.813355, 1.570796, 1.678255],accel_mss,speed_ms,0,blend_radius_m)
    |   movel([0.112766, -1.336699, -2.559921, -0.815769, 1.570796, 1.683562],accel_mss,speed_ms,0,blend_radius_m)
    |   movel([0.112766, -1.361858, -2.572418, -0.778114, 1.570796, 1.683562],accel_mss,speed_ms,0,blend_radius_m)
    |   speed_ms = 0.003
    |   movel([0.112766, -1.371669, -2.576969, -0.763751, 1.570796, 1.683562],accel_mss,speed_ms,0,blend_radius_m)
    |   speed_ms = 0.007
    |   movel([0.112640, -1.371423, -2.577139, -0.763827, 1.570796, 1.683436],accel_mss,speed_ms,0,blend_radius_m)
    |   movel([0.112664, -1.370800, -2.577571, -0.764018, 1.570796, 1.683461],accel_mss,speed_ms,0,blend_radius_m)
    |   movel([0.112748, -1.369984, -2.578135, -0.764270, 1.570796, 1.683545],accel_mss,speed_ms,0,blend_radius_m)
    |   movel([0.114064, -1.369651, -2.578365, -0.764373, 1.570796, 1.684861],accel_mss,speed_ms,0,blend_radius_m)
    |   movel([0.115040, -1.369430, -2.578518, -0.764442, 1.570796, 1.685836],accel_mss,speed_ms,0,blend_radius_m)
    |   movel([0.115513, -1.369409, -2.578532, -0.764448, 1.570796, 1.686309],accel_mss,speed_ms,0,blend_radius_m)
    |   movel([0.115676, -1.369559, -2.578429, -0.764401, 1.570796, 1.686472],accel_mss,speed_ms,0,blend_radius_m)
    |   movel([0.115615, -1.369869, -2.578214, -0.764305, 1.570796, 1.686411],accel_mss,speed_ms,0,blend_radius_m)
    |   movel([0.115514, -1.370131, -2.578033, -0.764225, 1.570796, 1.686311],accel_mss,speed_ms,0,blend_radius_m)
    |   movel([0.115438, -1.370635, -2.577685, -0.764069, 1.570796, 1.686234],accel_mss,speed_ms,0,blend_radius_m)
    |   movel([0.115115, -1.370976, -2.577449, -0.763964, 1.570796, 1.685911],accel_mss,speed_ms,0,blend_radius_m)
    |   movel([0.114542, -1.371299, -2.577225, -0.763865, 1.570796, 1.685338],accel_mss,speed_ms,0,blend_radius_m)
    |   movel([0.113790, -1.371559, -2.577045, -0.763785, 1.570796, 1.684586],accel_mss,speed_ms,0,blend_radius_m)
    |   movel([0.113081, -1.371719, -2.576934, -0.763736, 1.570796, 1.683877],accel_mss,speed_ms,0,blend_radius_m)
    |   movel([0.112766, -1.371669, -2.576969, -0.763751, 1.570796, 1.683562],accel_mss,speed_ms,0,blend_radius_m)
    |   speed_ms = 0.003
    |   movel([0.112766, -1.374985, -2.578469, -0.758934, 1.570796, 1.683562],accel_mss,speed_ms,0,blend_radius_m)
    |   speed_ms = 0.007
    |   movel([0.112640, -1.374740, -2.578640, -0.759009, 1.570796, 1.683436],accel_mss,speed_ms,0,blend_radius_m)
    |   movel([0.112664, -1.374119, -2.579072, -0.759198, 1.570796, 1.683461],accel_mss,speed_ms,0,blend_radius_m)
    |   movel([0.112748, -1.373305, -2.579638, -0.759446, 1.570796, 1.683545],accel_mss,speed_ms,0,blend_radius_m)
    |   movel([0.114064, -1.372973, -2.579869, -0.759547, 1.570796, 1.684861],accel_mss,speed_ms,0,blend_radius_m)
    |   movel([0.115040, -1.372752, -2.580022, -0.759615, 1.570796, 1.685836],accel_mss,speed_ms,0,blend_radius_m)
    |   movel([0.115513, -1.372732, -2.580036, -0.759621, 1.570796, 1.686309],accel_mss,speed_ms,0,blend_radius_m)
    |   movel([0.115676, -1.372881, -2.579932, -0.759576, 1.570796, 1.686472],accel_mss,speed_ms,0,blend_radius_m)
    |   movel([0.115615, -1.373191, -2.579717, -0.759481, 1.570796, 1.686411],accel_mss,speed_ms,0,blend_radius_m)
    |   movel([0.115514, -1.373452, -2.579536, -0.759401, 1.570796, 1.686311],accel_mss,speed_ms,0,blend_radius_m)
    |   movel([0.115438, -1.373954, -2.579187, -0.759248, 1.570796, 1.686234],accel_mss,speed_ms,0,blend_radius_m)
    |   movel([0.115115, -1.374294, -2.578951, -0.759144, 1.570796, 1.685911],accel_mss,speed_ms,0,blend_radius_m)
    |   movel([0.114542, -1.374617, -2.578726, -0.759046, 1.570796, 1.685338],accel_mss,speed_ms,0,blend_radius_m)
    |   movel([0.113790, -1.374876, -2.578545, -0.758968, 1.570796, 1.684586],accel_mss,speed_ms,0,blend_radius_m)
    |   movel([0.113081, -1.375035, -2.578434, -0.758919, 1.570796, 1.683877],accel_mss,speed_ms,0,blend_radius_m)
    |   movel([0.112766, -1.374985, -2.578469, -0.758934, 1.570796, 1.683562],accel_mss,speed_ms,0,blend_radius_m)
    |   speed_ms = 0.003
    |   movel([0.112766, -1.361858, -2.572418, -0.778114, 1.570796, 1.683562],accel_mss,speed_ms,0,blend_radius_m)
    |   speed_ms = 1.000
    |   movel([0.112766, -1.336699, -2.559921, -0.815769, 1.570796, 1.683562],accel_mss,speed_ms,0,blend_radius_m)
    |   movel([0.113433, -1.334323, -2.561482, -0.816584, 1.570796, 1.684229],accel_mss,speed_ms,0,blend_radius_m)
    |   movel([0.113433, -1.359522, -2.574009, -0.778858, 1.570796, 1.684229],accel_mss,speed_ms,0,blend_radius_m)
    |   speed_ms = 0.003
    |   movel([0.113433, -1.369351, -2.578572, -0.764466, 1.570796, 1.684229],accel_mss,speed_ms,0,blend_radius_m)
    |   speed_ms = 0.007
    |   movel([0.113200, -1.369116, -2.578734, -0.764539, 1.570796, 1.683996],accel_mss,speed_ms,0,blend_radius_m)
    |   movel([0.113209, -1.368786, -2.578962, -0.764641, 1.570796, 1.684005],accel_mss,speed_ms,0,blend_radius_m)
    |   movel([0.113200, -1.368460, -2.579187, -0.764743, 1.570796, 1.683996],accel_mss,speed_ms,0,blend_radius_m)
